  MoveL 5081 to (509.6, 509.6, 11.2) mm, rotated rx 0 ry 90 rz 0 deg; joints [-12.688, -27.246, 109.927, -16.748, -82.126, 51.332]
  Call Extruder(0.559)
  MoveL 5082 to (490.4, 509.6, 11.2) mm, rotated rx 0 ry 90 rz 0 deg; joints [-13.088, -27.603, 112.214, -17.082, -83.985, 50.809]
  MoveL 5083 to (490.4, 490.4, 11.2) mm, rotated rx 0 ry 90 rz 0 deg; joints [-11.303, -27.672, 112.704, -15.276, -84.344, 50.536]
  Call Extruder(0.199)
  MoveL 5084 to (497.23, 490.4, 11.2) mm, rotated rx 0 ry 90 rz 0 deg; joints [-11.177, -27.556, 111.894, -15.169, -83.672, 50.707]
  Call Extruder(0.010)
  MoveL 5085 to (497.58, 490.4, 11.2) mm, rotated rx 0 ry 90 rz 0 deg; joints [-11.17, -27.55, 111.853, -15.163, -83.637, 50.716]
  Call Extruder(0.007)
  MoveL 5086 to (497.58, 490.75, 11.2) mm, rotated rx 0 ry 90 rz 0 deg; joints [-11.203, -27.549, 111.844, -15.196, -83.631, 50.721]
  Call Extruder(0.035)
  MoveL 5087 to (497.57, 491.95, 11.2) mm, rotated rx 0 ry 90 rz 0 deg; joints [-11.314, -27.545, 111.816, -15.308, -83.611, 50.738]
  Call Extruder(0.007)
  MoveL 5088 to (497.58, 492.3, 11.2) mm, rotated rx 0 ry 90 rz 0 deg; joints [-11.346, -27.544, 111.808, -15.341, -83.605, 50.743]
  Set speed (120.0 mm/s)
  MoveL 5089 to (497.93, 492.3, 11.2) mm, rotated rx 0 ry 90 rz 0 deg; joints [-11.34, -27.537, 111.766, -15.336, -83.571, 50.752]
  Set speed (1000.0 mm/s)
  MoveL 5090 to (497.98, 492.3, 11.2) mm, rotated rx 0 ry 90 rz 0 deg; joints [-11.339, -27.536, 111.76, -15.335, -83.566, 50.753]
  Set speed (1000.0 mm/s)
  MoveL 5091 to (497.97, 493, 11.2) mm, rotated rx 0 ry 90 rz 0 deg; joints [-11.403, -27.534, 111.743, -15.4, -83.554, 50.764]
  Set speed (1000.0 mm/s)
  MoveL 5092 to (490.68, 490.68, 11.2) mm, rotated rx 0 ry 90 rz 0 deg; joints [-11.324, -27.666, 112.664, -15.298, -84.312, 50.546]
  Set speed (1000.0 mm/s)
  MoveL 5093 to (490.68, 490.68, 11.3) mm, rotated rx 0 ry 90 rz 0 deg; joints [-11.324, -27.677, 112.669, -15.298, -84.307, 50.548]
  Set speed (30.0 mm/s)
  Call Extruder(0.767)
  MoveL 5094 to (509.32, 509.32, 11.3) mm, rotated rx 0 ry 90 rz 0 deg; joints [-12.669, -27.264, 109.974, -16.727, -82.153, 51.321]
  MoveL 5095 to (509.44, 509.44, 11.3) mm, rotated rx 0 ry 90 rz 0 deg; joints [-12.677, -27.261, 109.956, -16.736, -82.139, 51.327]
  Set speed (120.0 mm/s)
  MoveL 5096 to (507.63, 502.27, 11.3) mm, rotated rx 0 ry 90 rz 0 deg; joints [-12.067, -27.328, 110.363, -16.108, -82.444, 51.156]
  Set speed (30.0 mm/s)
  Call Extruder(0.290)
  MoveL 5097 to (500.58, 509.32, 11.3) mm, rotated rx 0 ry 90 rz 0 deg; joints [-12.847, -27.433, 111.021, -16.874, -82.999, 51.086]
  Set speed (120.0 mm/s)
  MoveL 5098 to (499.42, 509.32, 11.3) mm, rotated rx 0 ry 90 rz 0 deg; joints [-12.872, -27.455, 111.159, -16.894, -83.111, 51.055]
  Set speed (30.0 mm/s)
  Call Extruder(0.360)
  MoveL 5099 to (490.68, 500.58, 11.3) mm, rotated rx 0 ry 90 rz 0 deg; joints [-12.247, -27.643, 112.425, -16.231, -84.127, 50.685]
  Set speed (120.0 mm/s)
  MoveL 5100 to (490.68, 499.42, 11.3) mm, rotated rx 0 ry 90 rz 0 deg; joints [-12.139, -27.647, 112.455, -16.122, -84.149, 50.668]
  Set speed (30.0 mm/s)
  Call Extruder(0.282)
  MoveL 5101 to (497.52, 492.58, 11.3) mm, rotated rx 0 ry 90 rz 0 deg; joints [-11.373, -27.554, 111.813, -15.368, -83.6, 50.747]
  MoveL 5102 to (497.64, 492.46, 11.3) mm, rotated rx 0 ry 90 rz 0 deg; joints [-11.359, -27.552, 111.801, -15.355, -83.59, 50.749]
  Set speed (120.0 mm/s)
  MoveL 5103 to (501.52, 492.33, 11.3) mm, rotated rx 0 ry 90 rz 0 deg; joints [-11.276, -27.483, 111.342, -15.283, -83.212, 50.844]
  Set speed (1000.0 mm/s)
  MoveL 5104 to (501.77, 491.87, 11.3) mm, rotated rx 0 ry 90 rz 0 deg; joints [-11.23, -27.48, 111.322, -15.237, -83.195, 50.844]
  Set speed (30.0 mm/s)
  Call Extruder(0.231)
  MoveL 5105 to (507.39, 497.49, 11.3) mm, rotated rx 0 ry 90 rz 0 deg; joints [-11.638, -27.353, 110.513, -15.671, -82.55, 51.072]
  MoveL 5106 to (507.51, 497.61, 11.3) mm, rotated rx 0 ry 90 rz 0 deg; joints [-11.647, -27.35, 110.495, -15.681, -82.536, 51.077]
  Set speed (120.0 mm/s)
  MoveL 5107 to (509.32, 490.68, 11.3) mm, rotated rx 0 ry 90 rz 0 deg; joints [-10.985, -27.341, 110.444, -15.015, -82.474, 51.011]
  Set speed (30.0 mm/s)
  Call Extruder(0.767)
  MoveL 5108 to (490.68, 509.32, 11.3) mm, rotated rx 0 ry 90 rz 0 deg; joints [-13.056, -27.61, 112.194, -17.051, -83.959, 50.814]
  MoveL 5109 to (490.56, 509.44, 11.3) mm, rotated rx 0 ry 90 rz 0 deg; joints [-13.07, -27.611, 112.205, -17.064, -83.968, 50.812]
  Set speed (120.0 mm/s)
  MoveL 5110 to (497.45, 492.37, 11.3) mm, rotated rx 0 ry 90 rz 0 deg; joints [-11.355, -27.556, 111.826, -15.35, -83.611, 50.743]
  Set speed (1000.0 mm/s)
  MoveL 5111 to (497.52, 492.3, 11.3) mm, rotated rx 0 ry 90 rz 0 deg; joints [-11.347, -27.555, 111.82, -15.342, -83.605, 50.743]
  Set speed (15.0 mm/s)
  Call Extruder(0.010)
  MoveL 5112 to (497.87, 492.3, 11.3) mm, rotated rx 0 ry 90 rz 0 deg; joints [-11.341, -27.549, 111.778, -15.337, -83.571, 50.752]
  Call Extruder(0.105)
  MoveL 5113 to (501.49, 492.3, 11.3) mm, rotated rx 0 ry 90 rz 0 deg; joints [-11.274, -27.484, 111.346, -15.281, -83.215, 50.843]
  Call Extruder(0.055)
  MoveL 5114 to (501.49, 490.4, 11.3) mm, rotated rx 0 ry 90 rz 0 deg; joints [-11.099, -27.491, 111.39, -15.104, -83.247, 50.815]
  Call Extruder(0.236)
  MoveL 5115 to (509.6, 490.4, 11.3) mm, rotated rx 0 ry 90 rz 0 deg; joints [-10.955, -27.337, 110.417, -14.985, -82.451, 51.013]
  Call Extruder(0.196)
  MoveL 5116 to (509.6, 497.15, 11.3) mm, rotated rx 0 ry 90 rz 0 deg; joints [-11.567, -27.31, 110.255, -15.607, -82.339, 51.122]
  Call Extruder(0.056)
  MoveL 5117 to (507.67, 497.15, 11.3) mm, rotated rx 0 ry 90 rz 0 deg; joints [-11.603, -27.348, 110.487, -15.636, -82.528, 51.073]
  Call Extruder(0.069)
  MoveL 5118 to (507.67, 499.52, 11.3) mm, rotated rx 0 ry 90 rz 0 deg; joints [-11.818, -27.339, 110.428, -15.854, -82.488, 51.112]
  Call Extruder(0.072)
  MoveL 5119 to (507.66, 501.99, 11.3) mm, rotated rx 0 ry 90 rz 0 deg; joints [-12.041, -27.329, 110.366, -16.082, -82.445, 51.153]
  Call Extruder(0.056)
  MoveL 5120 to (509.6, 502, 11.3) mm, rotated rx 0 ry 90 rz 0 deg; joints [-12.004, -27.29, 110.133, -16.052, -82.256, 51.203]
  Call Extruder(0.221)
  MoveL 5121 to (509.6, 509.6, 11.3) mm, rotated rx 0 ry 90 rz 0 deg; joints [-12.688, -27.257, 109.932, -16.748, -82.121, 51.334]
  Call Extruder(0.559)
  MoveL 5122 to (490.4, 509.6, 11.3) mm, rotated rx 0 ry 90 rz 0 deg; joints [-13.088, -27.613, 112.219, -17.082, -83.98, 50.811]
  MoveL 5123 to (490.4, 490.4, 11.3) mm, rotated rx 0 ry 90 rz 0 deg; joints [-11.303, -27.682, 112.709, -15.277, -84.339, 50.537]
  Call Extruder(0.197)
  MoveL 5124 to (497.17, 490.4, 11.3) mm, rotated rx 0 ry 90 rz 0 deg; joints [-11.178, -27.568, 111.906, -15.17, -83.672, 50.708]
  Call Extruder(0.010)
  MoveL 5125 to (497.52, 490.4, 11.3) mm, rotated rx 0 ry 90 rz 0 deg; joints [-11.171, -27.562, 111.864, -15.164, -83.638, 50.716]
  Call Extruder(0.007)
  MoveL 5126 to (497.52, 490.75, 11.3) mm, rotated rx 0 ry 90 rz 0 deg; joints [-11.204, -27.561, 111.856, -15.197, -83.632, 50.721]
  Call Extruder(0.035)
  MoveL 5127 to (497.52, 491.95, 11.3) mm, rotated rx 0 ry 90 rz 0 deg; joints [-11.315, -27.556, 111.828, -15.309, -83.611, 50.738]
  Call Extruder(0.007)
  MoveL 5128 to (497.52, 492.3, 11.3) mm, rotated rx 0 ry 90 rz 0 deg; joints [-11.347, -27.555, 111.82, -15.342, -83.605, 50.743]
  Set speed (120.0 mm/s)
  MoveL 5129 to (497.87, 492.3, 11.3) mm, rotated rx 0 ry 90 rz 0 deg; joints [-11.341, -27.549, 111.778, -15.337, -83.571, 50.752]
  Set speed (1000.0 mm/s)
  MoveL 5130 to (497.92, 492.3, 11.3) mm, rotated rx 0 ry 90 rz 0 deg; joints [-11.34, -27.548, 111.772, -15.336, -83.566, 50.753]
  Set speed (1000.0 mm/s)
  MoveL 5131 to (497.92, 493, 11.3) mm, rotated rx 0 ry 90 rz 0 deg; joints [-11.404, -27.546, 111.755, -15.401, -83.554, 50.764]
  Set speed (1000.0 mm/s)
  MoveL 5132 to (490.68, 490.68, 11.3) mm, rotated rx 0 ry 90 rz 0 deg; joints [-11.324, -27.677, 112.669, -15.298, -84.307, 50.548]
  Set speed (1000.0 mm/s)
  MoveL 5133 to (490.68, 490.68, 11.4) mm, rotated rx 0 ry 90 rz 0 deg; joints [-11.324, -27.688, 112.675, -15.299, -84.301, 50.549]
  Set speed (30.0 mm/s)
  Call Extruder(0.767)
  MoveL 5134 to (509.32, 509.32, 11.4) mm, rotated rx 0 ry 90 rz 0 deg; joints [-12.669, -27.274, 109.979, -16.727, -82.148, 51.323]
  MoveL 5135 to (509.44, 509.44, 11.4) mm, rotated rx 0 ry 90 rz 0 deg; joints [-12.677, -27.271, 109.961, -16.736, -82.134, 51.328]
  Set speed (120.0 mm/s)
  MoveL 5136 to (507.57, 502.33, 11.4) mm, rotated rx 0 ry 90 rz 0 deg; joints [-12.073, -27.34, 110.374, -16.114, -82.443, 51.157]
  Set speed (30.0 mm/s)
  Call Extruder(0.288)
  MoveL 5137 to (500.58, 509.32, 11.4) mm, rotated rx 0 ry 90 rz 0 deg; joints [-12.847, -27.444, 111.026, -16.874, -82.994, 51.088]
  Set speed (120.0 mm/s)
  MoveL 5138 to (499.42, 509.32, 11.4) mm, rotated rx 0 ry 90 rz 0 deg; joints [-12.872, -27.465, 111.164, -16.894, -83.106, 51.056]
  Set speed (30.0 mm/s)
  Call Extruder(0.360)
  MoveL 5139 to (490.68, 500.58, 11.4) mm, rotated rx 0 ry 90 rz 0 deg; joints [-12.247, -27.653, 112.431, -16.231, -84.122, 50.686]
  Set speed (120.0 mm/s)
  MoveL 5140 to (490.68, 499.42, 11.4) mm, rotated rx 0 ry 90 rz 0 deg; joints [-12.139, -27.658, 112.46, -16.122, -84.144, 50.67]
  Set speed (30.0 mm/s)
  Call Extruder(0.282)
  MoveL 5141 to (497.52, 492.58, 11.4) mm, rotated rx 0 ry 90 rz 0 deg; joints [-11.373, -27.565, 111.818, -15.368, -83.595, 50.749]
  MoveL 5142 to (497.64, 492.46, 11.4) mm, rotated rx 0 ry 90 rz 0 deg; joints [-11.359, -27.563, 111.806, -15.355, -83.585, 50.75]
  Set speed (120.0 mm/s)
  MoveL 5143 to (501.59, 492.33, 11.4) mm, rotated rx 0 ry 90 rz 0 deg; joints [-11.275, -27.493, 111.339, -15.282, -83.2, 50.847]
  Set speed (1000.0 mm/s)
  MoveL 5144 to (501.84, 491.94, 11.4) mm, rotated rx 0 ry 90 rz 0 deg; joints [-11.234, -27.489, 111.318, -15.242, -83.182, 50.848]
  Set speed (30.0 mm/s)
  Call Extruder(0.228)
  MoveL 5145 to (507.39, 497.49, 11.4) mm, rotated rx 0 ry 90 rz 0 deg; joints [-11.638, -27.363, 110.518, -15.671, -82.545, 51.073]
  MoveL 5146 to (507.51, 497.61, 11.4) mm, rotated rx 0 ry 90 rz 0 deg; joints [-11.647, -27.36, 110.5, -15.681, -82.531, 51.078]
  Set speed (120.0 mm/s)
  MoveL 5147 to (509.32, 490.68, 11.4) mm, rotated rx 0 ry 90 rz 0 deg; joints [-10.985, -27.352, 110.449, -15.015, -82.469, 51.012]
  Set speed (30.0 mm/s)
  Call Extruder(0.767)
  MoveL 5148 to (490.68, 509.32, 11.4) mm, rotated rx 0 ry 90 rz 0 deg; joints [-13.056, -27.62, 112.199, -17.051, -83.953, 50.816]
  MoveL 5149 to (490.56, 509.44, 11.4) mm, rotated rx 0 ry 90 rz 0 deg; joints [-13.07, -27.622, 112.21, -17.065, -83.963, 50.814]
  Set speed (120.0 mm/s)
  MoveL 5150 to (507.6, 499.64, 11.4) mm, rotated rx 0 ry 90 rz 0 deg; joints [-11.83, -27.35, 110.439, -15.867, -82.487, 51.114]
  Set speed (1000.0 mm/s)
  MoveL 5151 to (507.67, 499.57, 11.4) mm, rotated rx 0 ry 90 rz 0 deg; joints [-11.822, -27.349, 110.432, -15.859, -82.482, 51.114]
  Set speed (15.0 mm/s)
  Call Extruder(0.010)
  MoveL 5152 to (508.02, 499.57, 11.4) mm, rotated rx 0 ry 90 rz 0 deg; joints [-11.816, -27.342, 110.39, -15.854, -82.447, 51.123]
  Call Extruder(0.046)
  MoveL 5153 to (509.6, 499.57, 11.4) mm, rotated rx 0 ry 90 rz 0 deg; joints [-11.786, -27.311, 110.2, -15.829, -82.293, 51.163]
  Call Extruder(0.000)
  MoveL 5154 to (509.6, 499.58, 11.4) mm, rotated rx 0 ry 90 rz 0 deg; joints [-11.786, -27.311, 110.199, -15.83, -82.293, 51.164]
  Call Extruder(0.046)
  MoveL 5155 to (508.02, 499.58, 11.4) mm, rotated rx 0 ry 90 rz 0 deg; joints [-11.816, -27.342, 110.39, -15.854, -82.447, 51.123]
  Call Extruder(0.010)
  MoveL 5156 to (507.67, 499.58, 11.4) mm, rotated rx 0 ry 90 rz 0 deg; joints [-11.823, -27.349, 110.432, -15.86, -82.482, 51.114]
  Call Extruder(0.007)
  MoveL 5157 to (507.67, 499.93, 11.4) mm, rotated rx 0 ry 90 rz 0 deg; joints [-11.854, -27.348, 110.423, -15.892, -82.475, 51.12]
  Call Extruder(0.062)
  MoveL 5158 to (507.66, 502.05, 11.4) mm, rotated rx 0 ry 90 rz 0 deg; joints [-12.046, -27.339, 110.37, -16.087, -82.439, 51.155]
  Call Extruder(0.056)
  MoveL 5159 to (509.6, 502.05, 11.4) mm, rotated rx 0 ry 90 rz 0 deg; joints [-12.009, -27.301, 110.137, -16.057, -82.25, 51.205]
  Call Extruder(0.220)
  MoveL 5160 to (509.6, 509.6, 11.4) mm, rotated rx 0 ry 90 rz 0 deg; joints [-12.688, -27.267, 109.938, -16.748, -82.115, 51.335]
  Call Extruder(0.559)
  MoveL 5161 to (490.4, 509.6, 11.4) mm, rotated rx 0 ry 90 rz 0 deg; joints [-13.088, -27.624, 112.224, -17.082, -83.975, 50.812]
  MoveL 5162 to (490.4, 490.4, 11.4) mm, rotated rx 0 ry 90 rz 0 deg; joints [-11.303, -27.693, 112.714, -15.277, -84.334, 50.538]
  Call Extruder(0.195)
  MoveL 5163 to (497.11, 490.4, 11.4) mm, rotated rx 0 ry 90 rz 0 deg; joints [-11.179, -27.58, 111.918, -15.171, -83.672, 50.708]
  Call Extruder(0.010)
  MoveL 5164 to (497.46, 490.4, 11.4) mm, rotated rx 0 ry 90 rz 0 deg; joints [-11.172, -27.573, 111.876, -15.165, -83.638, 50.716]
  Call Extruder(0.007)
  MoveL 5165 to (497.46, 490.75, 11.4) mm, rotated rx 0 ry 90 rz 0 deg; joints [-11.205, -27.572, 111.868, -15.198, -83.632, 50.721]
  Call Extruder(0.035)
  MoveL 5166 to (497.46, 491.95, 11.4) mm, rotated rx 0 ry 90 rz 0 deg; joints [-11.316, -27.568, 111.84, -15.31, -83.612, 50.738]
  Call Extruder(0.010)
  MoveL 5167 to (497.46, 492.3, 11.4) mm, rotated rx 0 ry 90 rz 0 deg; joints [-11.348, -27.567, 111.831, -15.343, -83.606, 50.743]
  Call Extruder(0.007)
  MoveL 5168 to (497.81, 492.3, 11.4) mm, rotated rx 0 ry 90 rz 0 deg; joints [-11.342, -27.561, 111.79, -15.338, -83.571, 50.752]
  Call Extruder(0.109)
  MoveL 5169 to (501.56, 492.3, 11.4) mm, rotated rx 0 ry 90 rz 0 deg; joints [-11.272, -27.493, 111.343, -15.28, -83.203, 50.846]
  Call Extruder(0.055)
  MoveL 5170 to (501.56, 490.4, 11.4) mm, rotated rx 0 ry 90 rz 0 deg; joints [-11.098, -27.5, 111.388, -15.103, -83.235, 50.818]
  Call Extruder(0.234)
  MoveL 5171 to (509.6, 490.4, 11.4) mm, rotated rx 0 ry 90 rz 0 deg; joints [-10.955, -27.347, 110.422, -14.985, -82.445, 51.015]
  Call Extruder(0.195)
  MoveL 5172 to (509.6, 497.09, 11.4) mm, rotated rx 0 ry 90 rz 0 deg; joints [-11.561, -27.321, 110.261, -15.601, -82.335, 51.122]
  Call Extruder(0.056)
  MoveL 5173 to (507.67, 497.09, 11.4) mm, rotated rx 0 ry 90 rz 0 deg; joints [-11.597, -27.359, 110.494, -15.631, -82.524, 51.074]
  Call Extruder(0.062)
  MoveL 5174 to (507.67, 499.22, 11.4) mm, rotated rx 0 ry 90 rz 0 deg; joints [-11.79, -27.351, 110.441, -15.827, -82.488, 51.108]
  Call Extruder(0.007)
  MoveL 5175 to (507.67, 499.57, 11.4) mm, rotated rx 0 ry 90 rz 0 deg; joints [-11.822, -27.349, 110.432, -15.859, -82.482, 51.114]
  Set speed (120.0 mm/s)
  MoveL 5176 to (508.02, 499.57, 11.4) mm, rotated rx 0 ry 90 rz 0 deg; joints [-11.816, -27.342, 110.39, -15.854, -82.447, 51.123]
  Set speed (1000.0 mm/s)
  MoveL 5177 to (508.07, 499.57, 11.4) mm, rotated rx 0 ry 90 rz 0 deg; joints [-11.815, -27.341, 110.384, -15.853, -82.443, 51.124]
  Set speed (1000.0 mm/s)
  MoveL 5178 to (506.97, 500.27, 11.4) mm, rotated rx 0 ry 90 rz 0 deg; joints [-11.899, -27.36, 110.499, -15.934, -82.538, 51.108]
  Set speed (1000.0 mm/s)
  MoveL 5179 to (490.68, 490.68, 11.4) mm, rotated rx 0 ry 90 rz 0 deg; joints [-11.324, -27.688, 112.675, -15.299, -84.301, 50.549]
  Set speed (1000.0 mm/s)
  MoveL 5180 to (490.68, 490.68, 11.5) mm, rotated rx 0 ry 90 rz 0 deg; joints [-11.324, -27.698, 112.68, -15.299, -84.296, 50.551]
  Set speed (30.0 mm/s)
  Call Extruder(0.767)
  MoveL 5181 to (509.32, 509.32, 11.5) mm, rotated rx 0 ry 90 rz 0 deg; joints [-12.669, -27.285, 109.984, -16.727, -82.143, 51.324]
  MoveL 5182 to (509.44, 509.44, 11.5) mm, rotated rx 0 ry 90 rz 0 deg; joints [-12.677, -27.282, 109.966, -16.737, -82.129, 51.33]
  Set speed (120.0 mm/s)
  MoveL 5183 to (507.51, 502.39, 11.5) mm, rotated rx 0 ry 90 rz 0 deg; joints [-12.08, -27.351, 110.384, -16.121, -82.442, 51.158]
  Set speed (30.0 mm/s)
  Call Extruder(0.285)
  MoveL 5184 to (500.58, 509.32, 11.5) mm, rotated rx 0 ry 90 rz 0 deg; joints [-12.847, -27.454, 111.031, -16.874, -82.988, 51.089]
  Set speed (120.0 mm/s)
  MoveL 5185 to (499.42, 509.32, 11.5) mm, rotated rx 0 ry 90 rz 0 deg; joints [-12.872, -27.476, 111.169, -16.895, -83.101, 51.058]
  Set speed (30.0 mm/s)
  Call Extruder(0.360)
  MoveL 5186 to (490.68, 500.58, 11.5) mm, rotated rx 0 ry 90 rz 0 deg; joints [-12.247, -27.664, 112.436, -16.232, -84.117, 50.688]
  Set speed (120.0 mm/s)
  MoveL 5187 to (490.68, 499.42, 11.5) mm, rotated rx 0 ry 90 rz 0 deg; joints [-12.139, -27.668, 112.465, -16.123, -84.138, 50.671]
  Set speed (30.0 mm/s)
  Call Extruder(0.282)
  MoveL 5188 to (497.52, 492.58, 11.5) mm, rotated rx 0 ry 90 rz 0 deg; joints [-11.373, -27.575, 111.823, -15.368, -83.59, 50.75]
  MoveL 5189 to (497.64, 492.46, 11.5) mm, rotated rx 0 ry 90 rz 0 deg; joints [-11.359, -27.574, 111.811, -15.355, -83.58, 50.752]
  Set speed (120.0 mm/s)
  MoveL 5190 to (501.65, 492.33, 11.5) mm, rotated rx 0 ry 90 rz 0 deg; joints [-11.273, -27.502, 111.337, -15.281, -83.189, 50.85]
  Set speed (1000.0 mm/s)
  MoveL 5191 to (501.9, 492, 11.5) mm, rotated rx 0 ry 90 rz 0 deg; joints [-11.239, -27.498, 111.314, -15.247, -83.17, 50.852]
  Set speed (30.0 mm/s)
  Call Extruder(0.226)
  MoveL 5192 to (507.39, 497.49, 11.5) mm, rotated rx 0 ry 90 rz 0 deg; joints [-11.638, -27.374, 110.523, -15.672, -82.54, 51.075]
  MoveL 5193 to (507.51, 497.61, 11.5) mm, rotated rx 0 ry 90 rz 0 deg; joints [-11.647, -27.371, 110.506, -15.681, -82.526, 51.08]
  Set speed (120.0 mm/s)
  MoveL 5194 to (509.32, 490.68, 11.5) mm, rotated rx 0 ry 90 rz 0 deg; joints [-10.985, -27.362, 110.454, -15.015, -82.463, 51.014]
  Set speed (30.0 mm/s)
  Call Extruder(0.767)
  MoveL 5195 to (490.68, 509.32, 11.5) mm, rotated rx 0 ry 90 rz 0 deg; joints [-13.056, -27.631, 112.204, -17.051, -83.948, 50.817]
  MoveL 5196 to (490.56, 509.44, 11.5) mm, rotated rx 0 ry 90 rz 0 deg; joints [-13.07, -27.633, 112.216, -17.065, -83.958, 50.816]
  Set speed (120.0 mm/s)
  MoveL 5197 to (507.6, 499.56, 11.5) mm, rotated rx 0 ry 90 rz 0 deg; joints [-11.823, -27.361, 110.446, -15.86, -82.484, 51.114]
  Set speed (1000.0 mm/s)
  MoveL 5198 to (507.67, 499.63, 11.5) mm, rotated rx 0 ry 90 rz 0 deg; joints [-11.828, -27.359, 110.436, -15.865, -82.476, 51.117]
  Set speed (15.0 mm/s)
  Call Extruder(0.010)
  MoveL 5199 to (507.67, 499.98, 11.5) mm, rotated rx 0 ry 90 rz 0 deg; joints [-11.859, -27.358, 110.427, -15.897, -82.469, 51.122]
  Call Extruder(0.062)
  MoveL 5200 to (507.67, 502.11, 11.5) mm, rotated rx 0 ry 90 rz 0 deg; joints [-12.051, -27.349, 110.373, -16.092, -82.432, 51.157]
  Call Extruder(0.056)
  MoveL 5201 to (509.6, 502.11, 11.5) mm, rotated rx 0 ry 90 rz 0 deg; joints [-12.015, -27.311, 110.14, -16.063, -82.244, 51.207]
  Call Extruder(0.218)
  MoveL 5202 to (509.6, 509.6, 11.5) mm, rotated rx 0 ry 90 rz 0 deg; joints [-12.688, -27.278, 109.943, -16.748, -82.11, 51.337]
  Call Extruder(0.559)
  MoveL 5203 to (490.4, 509.6, 11.5) mm, rotated rx 0 ry 90 rz 0 deg; joints [-13.088, -27.635, 112.23, -17.082, -83.97, 50.814]
  MoveL 5204 to (490.4, 490.4, 11.5) mm, rotated rx 0 ry 90 rz 0 deg; joints [-11.303, -27.704, 112.719, -15.277, -84.329, 50.54]
  Call Extruder(0.204)
  MoveL 5205 to (497.41, 490.4, 11.5) mm, rotated rx 0 ry 90 rz 0 deg; joints [-11.173, -27.585, 111.888, -15.166, -83.638, 50.716]
  Call Extruder(0.045)
  MoveL 5206 to (497.41, 491.95, 11.5) mm, rotated rx 0 ry 90 rz 0 deg; joints [-11.317, -27.58, 111.852, -15.311, -83.612, 50.738]
  Call Extruder(0.010)
  MoveL 5207 to (497.41, 492.3, 11.5) mm, rotated rx 0 ry 90 rz 0 deg; joints [-11.349, -27.578, 111.843, -15.344, -83.606, 50.743]
  Call Extruder(0.007)
  MoveL 5208 to (497.76, 492.3, 11.5) mm, rotated rx 0 ry 90 rz 0 deg; joints [-11.343, -27.572, 111.802, -15.339, -83.571, 50.752]
  Call Extruder(0.112)
  MoveL 5209 to (501.62, 492.3, 11.5) mm, rotated rx 0 ry 90 rz 0 deg; joints [-11.271, -27.503, 111.341, -15.279, -83.192, 50.849]
  Call Extruder(0.055)
  MoveL 5210 to (501.62, 490.4, 11.5) mm, rotated rx 0 ry 90 rz 0 deg; joints [-11.097, -27.509, 111.385, -15.102, -83.224, 50.821]
  Call Extruder(0.232)
  MoveL 5211 to (509.6, 490.4, 11.5) mm, rotated rx 0 ry 90 rz 0 deg; joints [-10.955, -27.358, 110.427, -14.985, -82.44, 51.016]
  Call Extruder(0.193)
  MoveL 5212 to (509.6, 497.03, 11.5) mm, rotated rx 0 ry 90 rz 0 deg; joints [-11.556, -27.332, 110.268, -15.596, -82.331, 51.123]
  Call Extruder(0.056)
  MoveL 5213 to (507.67, 497.03, 11.5) mm, rotated rx 0 ry 90 rz 0 deg; joints [-11.592, -27.37, 110.501, -15.626, -82.52, 51.074]
  Call Extruder(0.062)
  MoveL 5214 to (507.67, 499.16, 11.5) mm, rotated rx 0 ry 90 rz 0 deg; joints [-11.785, -27.361, 110.448, -15.822, -82.483, 51.109]
  Call Extruder(0.010)
  MoveL 5215 to (507.67, 499.51, 11.5) mm, rotated rx 0 ry 90 rz 0 deg; joints [-11.817, -27.36, 110.439, -15.854, -82.477, 51.115]
  Call Extruder(0.007)
  MoveL 5216 to (508.02, 499.51, 11.5) mm, rotated rx 0 ry 90 rz 0 deg; joints [-11.81, -27.353, 110.397, -15.849, -82.443, 51.124]
  Call Extruder(0.046)
  MoveL 5217 to (509.6, 499.51, 11.5) mm, rotated rx 0 ry 90 rz 0 deg; joints [-11.78, -27.322, 110.206, -15.824, -82.289, 51.164]
  Call Extruder(0.004)
  MoveL 5218 to (509.6, 499.64, 11.5) mm, rotated rx 0 ry 90 rz 0 deg; joints [-11.792, -27.321, 110.203, -15.836, -82.287, 51.166]
  Call Extruder(0.046)
  MoveL 5219 to (508.02, 499.63, 11.5) mm, rotated rx 0 ry 90 rz 0 deg; joints [-11.821, -27.352, 110.394, -15.86, -82.441, 51.126]
  Call Extruder(0.007)
  MoveL 5220 to (507.67, 499.63, 11.5) mm, rotated rx 0 ry 90 rz 0 deg; joints [-11.828, -27.359, 110.436, -15.865, -82.476, 51.117]
  Set speed (120.0 mm/s)
  MoveL 5221 to (507.67, 499.98, 11.5) mm, rotated rx 0 ry 90 rz 0 deg; joints [-11.859, -27.358, 110.427, -15.897, -82.469, 51.122]
  Set speed (1000.0 mm/s)
  MoveL 5222 to (507.67, 500.03, 11.5) mm, rotated rx 0 ry 90 rz 0 deg; joints [-11.864, -27.358, 110.426, -15.902, -82.469, 51.123]
  Set speed (1000.0 mm/s)
  MoveL 5223 to (506.97, 500.03, 11.5) mm, rotated rx 0 ry 90 rz 0 deg; joints [-11.877, -27.371, 110.51, -15.913, -82.537, 51.105]
  Set speed (1000.0 mm/s)
  MoveL 5224 to (490.68, 490.68, 11.5) mm, rotated rx 0 ry 90 rz 0 deg; joints [-11.324, -27.698, 112.68, -15.299, -84.296, 50.551]
  Set speed (1000.0 mm/s)
  MoveL 5225 to (490.68, 490.68, 11.6) mm, rotated rx 0 ry 90 rz 0 deg; joints [-11.324, -27.709, 112.685, -15.299, -84.291, 50.552]
  Set speed (30.0 mm/s)
  Call Extruder(0.767)
  MoveL 5226 to (509.32, 509.32, 11.6) mm, rotated rx 0 ry 90 rz 0 deg; joints [-12.669, -27.295, 109.989, -16.728, -82.138, 51.326]
  MoveL 5227 to (509.44, 509.44, 11.6) mm, rotated rx 0 ry 90 rz 0 deg; joints [-12.677, -27.292, 109.971, -16.737, -82.123, 51.331]
  Set speed (120.0 mm/s)
  MoveL 5228 to (507.46, 502.44, 11.6) mm, rotated rx 0 ry 90 rz 0 deg; joints [-12.086, -27.362, 110.395, -16.127, -82.442, 51.159]
  Set speed (30.0 mm/s)
  Call Extruder(0.283)
  MoveL 5229 to (500.58, 509.32, 11.6) mm, rotated rx 0 ry 90 rz 0 deg; joints [-12.847, -27.465, 111.036, -16.875, -82.983, 51.091]
  Set speed (120.0 mm/s)
  MoveL 5230 to (499.42, 509.32, 11.6) mm, rotated rx 0 ry 90 rz 0 deg; joints [-12.872, -27.487, 111.174, -16.895, -83.096, 51.059]
  Set speed (30.0 mm/s)
  Call Extruder(0.360)
  MoveL 5231 to (490.68, 500.58, 11.6) mm, rotated rx 0 ry 90 rz 0 deg; joints [-12.247, -27.675, 112.441, -16.232, -84.112, 50.689]
  Set speed (120.0 mm/s)
  MoveL 5232 to (490.68, 499.42, 11.6) mm, rotated rx 0 ry 90 rz 0 deg; joints [-12.139, -27.679, 112.471, -16.123, -84.133, 50.673]
  Set speed (30.0 mm/s)
  Call Extruder(0.282)
  MoveL 5233 to (497.52, 492.58, 11.6) mm, rotated rx 0 ry 90 rz 0 deg; joints [-11.373, -27.586, 111.828, -15.369, -83.585, 50.752]
  MoveL 5234 to (497.64, 492.46, 11.6) mm, rotated rx 0 ry 90 rz 0 deg; joints [-11.359, -27.584, 111.817, -15.355, -83.575, 50.753]
  Set speed (120.0 mm/s)
  MoveL 5235 to (501.71, 492.33, 11.6) mm, rotated rx 0 ry 90 rz 0 deg; joints [-11.272, -27.511, 111.334, -15.28, -83.177, 50.853]
  Set speed (1000.0 mm/s)
  MoveL 5236 to (501.96, 492.06, 11.6) mm, rotated rx 0 ry 90 rz 0 deg; joints [-11.244, -27.508, 111.31, -15.252, -83.157, 50.856]
  Set speed (30.0 mm/s)
  Call Extruder(0.223)
  MoveL 5237 to (507.39, 497.49, 11.6) mm, rotated rx 0 ry 90 rz 0 deg; joints [-11.638, -27.384, 110.528, -15.672, -82.534, 51.076]
  MoveL 5238 to (507.51, 497.61, 11.6) mm, rotated rx 0 ry 90 rz 0 deg; joints [-11.647, -27.381, 110.51, -15.681, -82.52, 51.081]
  Set speed (120.0 mm/s)
  MoveL 5239 to (509.32, 490.68, 11.6) mm, rotated rx 0 ry 90 rz 0 deg; joints [-10.985, -27.373, 110.46, -15.015, -82.458, 51.015]
  Set speed (30.0 mm/s)
  Call Extruder(0.767)
  MoveL 5240 to (490.68, 509.32, 11.6) mm, rotated rx 0 ry 90 rz 0 deg; joints [-13.056, -27.642, 112.21, -17.051, -83.943, 50.819]
  MoveL 5241 to (490.56, 509.44, 11.6) mm, rotated rx 0 ry 90 rz 0 deg; joints [-13.07, -27.643, 112.221, -17.065, -83.952, 50.817]
  Set speed (120.0 mm/s)
  MoveL 5242 to (507.6, 499.52, 11.6) mm, rotated rx 0 ry 90 rz 0 deg; joints [-11.819, -27.372, 110.452, -15.856, -82.479, 51.115]
  Set speed (1000.0 mm/s)
  MoveL 5243 to (507.67, 499.46, 11.6) mm, rotated rx 0 ry 90 rz 0 deg; joints [-11.812, -27.371, 110.445, -15.849, -82.473, 51.115]
  Set speed (15.0 mm/s)
  Call Extruder(0.010)
  MoveL 5244 to (508.02, 499.45, 11.6) mm, rotated rx 0 ry 90 rz 0 deg; joints [-11.805, -27.364, 110.404, -15.843, -82.439, 51.124]
  Call Extruder(0.046)
  MoveL 5245 to (509.6, 499.45, 11.6) mm, rotated rx 0 ry 90 rz 0 deg; joints [-11.775, -27.332, 110.213, -15.819, -82.285, 51.164]
  Call Extruder(0.007)
  MoveL 5246 to (509.6, 499.69, 11.6) mm, rotated rx 0 ry 90 rz 0 deg; joints [-11.796, -27.331, 110.207, -15.841, -82.281, 51.168]
  Call Extruder(0.031)
  MoveL 5247 to (508.02, 499.69, 11.6) mm, rotated rx 0 ry 90 rz 0 deg; joints [-11.826, -27.363, 110.398, -15.865, -82.435, 51.128]
  Call Extruder(0.007)
  MoveL 5248 to (507.67, 499.69, 11.6) mm, rotated rx 0 ry 90 rz 0 deg; joints [-11.833, -27.37, 110.44, -15.87, -82.469, 51.119]
  Call Extruder(0.007)
  MoveL 5249 to (507.67, 500.04, 11.6) mm, rotated rx 0 ry 90 rz 0 deg; joints [-11.865, -27.368, 110.431, -15.903, -82.463, 51.125]
  Call Extruder(0.062)
  MoveL 5250 to (507.67, 502.16, 11.6) mm, rotated rx 0 ry 90 rz 0 deg; joints [-12.057, -27.359, 110.377, -16.098, -82.426, 51.16]
  Call Extruder(0.056)
  MoveL 5251 to (509.6, 502.17, 11.6) mm, rotated rx 0 ry 90 rz 0 deg; joints [-12.02, -27.321, 110.144, -16.068, -82.238, 51.21]
  Call Extruder(0.216)
  MoveL 5252 to (509.6, 509.6, 11.6) mm, rotated rx 0 ry 90 rz 0 deg; joints [-12.688, -27.288, 109.948, -16.749, -82.105, 51.338]
  Call Extruder(0.559)
  MoveL 5253 to (490.4, 509.6, 11.6) mm, rotated rx 0 ry 90 rz 0 deg; joints [-13.088, -27.645, 112.235, -17.083, -83.964, 50.815]
  MoveL 5254 to (490.4, 490.4, 11.6) mm, rotated rx 0 ry 90 rz 0 deg; joints [-11.303, -27.715, 112.725, -15.277, -84.323, 50.541]
  Call Extruder(0.192)
  MoveL 5255 to (497, 490.4, 11.6) mm, rotated rx 0 ry 90 rz 0 deg; joints [-11.181, -27.603, 111.942, -15.173, -83.673, 50.708]
  Call Extruder(0.010)
  MoveL 5256 to (497.35, 490.4, 11.6) mm, rotated rx 0 ry 90 rz 0 deg; joints [-11.175, -27.597, 111.9, -15.167, -83.639, 50.716]
  Call Extruder(0.007)
  MoveL 5257 to (497.35, 490.75, 11.6) mm, rotated rx 0 ry 90 rz 0 deg; joints [-11.207, -27.595, 111.892, -15.2, -83.633, 50.721]
  Call Extruder(0.035)
  MoveL 5258 to (497.35, 491.95, 11.6) mm, rotated rx 0 ry 90 rz 0 deg; joints [-11.318, -27.591, 111.864, -15.312, -83.612, 50.738]
  Call Extruder(0.010)
  MoveL 5259 to (497.35, 492.3, 11.6) mm, rotated rx 0 ry 90 rz 0 deg; joints [-11.35, -27.59, 111.855, -15.345, -83.606, 50.743]
  Call Extruder(0.007)
  MoveL 5260 to (497.7, 492.3, 11.6) mm, rotated rx 0 ry 90 rz 0 deg; joints [-11.344, -27.584, 111.814, -15.34, -83.572, 50.752]
  Call Extruder(0.116)
  MoveL 5261 to (501.68, 492.3, 11.6) mm, rotated rx 0 ry 90 rz 0 deg; joints [-11.27, -27.512, 111.338, -15.278, -83.18, 50.852]
  Call Extruder(0.055)
  MoveL 5262 to (501.68, 490.4, 11.6) mm, rotated rx 0 ry 90 rz 0 deg; joints [-11.096, -27.519, 111.383, -15.101, -83.212, 50.824]
  Call Extruder(0.230)
  MoveL 5263 to (509.6, 490.4, 11.6) mm, rotated rx 0 ry 90 rz 0 deg; joints [-10.955, -27.368, 110.432, -14.986, -82.435, 51.018]
  Call Extruder(0.191)
  MoveL 5264 to (509.6, 496.97, 11.6) mm, rotated rx 0 ry 90 rz 0 deg; joints [-11.551, -27.343, 110.275, -15.591, -82.327, 51.123]
  Call Extruder(0.056)
  MoveL 5265 to (507.67, 496.97, 11.6) mm, rotated rx 0 ry 90 rz 0 deg; joints [-11.587, -27.381, 110.507, -15.62, -82.516, 51.075]
  Call Extruder(0.062)
  MoveL 5266 to (507.67, 499.11, 11.6) mm, rotated rx 0 ry 90 rz 0 deg; joints [-11.78, -27.372, 110.454, -15.817, -82.479, 51.11]
  Call Extruder(0.007)
  MoveL 5267 to (507.67, 499.46, 11.6) mm, rotated rx 0 ry 90 rz 0 deg; joints [-11.812, -27.371, 110.445, -15.849, -82.473, 51.115]
  Set speed (120.0 mm/s)
  MoveL 5268 to (508.02, 499.45, 11.6) mm, rotated rx 0 ry 90 rz 0 deg; joints [-11.805, -27.364, 110.404, -15.843, -82.439, 51.124]
  Set speed (1000.0 mm/s)
  MoveL 5269 to (508.07, 499.45, 11.6) mm, rotated rx 0 ry 90 rz 0 deg; joints [-11.804, -27.363, 110.397, -15.843, -82.434, 51.125]
  Set speed (1000.0 mm/s)
  MoveL 5270 to (506.97, 500.15, 11.6) mm, rotated rx 0 ry 90 rz 0 deg; joints [-11.888, -27.381, 110.512, -15.924, -82.53, 51.109]
  Set speed (1000.0 mm/s)
  MoveL 5271 to (490.68, 490.68, 11.6) mm, rotated rx 0 ry 90 rz 0 deg; joints [-11.324, -27.709, 112.685, -15.299, -84.291, 50.552]
  Set speed (1000.0 mm/s)
  MoveL 5272 to (490.68, 490.68, 11.7) mm, rotated rx 0 ry 90 rz 0 deg; joints [-11.324, -27.72, 112.69, -15.299, -84.286, 50.554]
  Set speed (30.0 mm/s)
  Call Extruder(0.767)
  MoveL 5273 to (509.32, 509.32, 11.7) mm, rotated rx 0 ry 90 rz 0 deg; joints [-12.669, -27.306, 109.994, -16.728, -82.133, 51.327]
  MoveL 5274 to (509.44, 509.44, 11.7) mm, rotated rx 0 ry 90 rz 0 deg; joints [-12.677, -27.303, 109.976, -16.737, -82.118, 51.333]
  Set speed (120.0 mm/s)
  MoveL 5275 to (507.4, 502.5, 11.7) mm, rotated rx 0 ry 90 rz 0 deg; joints [-12.092, -27.374, 110.405, -16.133, -82.441, 51.16]
  Set speed (30.0 mm/s)
  Call Extruder(0.281)
  MoveL 5276 to (500.58, 509.32, 11.7) mm, rotated rx 0 ry 90 rz 0 deg; joints [-12.847, -27.476, 111.041, -16.875, -82.978, 51.092]
  Set speed (120.0 mm/s)
  MoveL 5277 to (499.42, 509.32, 11.7) mm, rotated rx 0 ry 90 rz 0 deg; joints [-12.872, -27.497, 111.179, -16.895, -83.09, 51.061]
  Set speed (30.0 mm/s)
  Call Extruder(0.360)
  MoveL 5278 to (490.68, 500.58, 11.7) mm, rotated rx 0 ry 90 rz 0 deg; joints [-12.247, -27.685, 112.446, -16.232, -84.106, 50.691]
  Set speed (120.0 mm/s)
  MoveL 5279 to (490.68, 499.42, 11.7) mm, rotated rx 0 ry 90 rz 0 deg; joints [-12.139, -27.69, 112.476, -16.123, -84.128, 50.674]
  Set speed (30.0 mm/s)
  Call Extruder(0.282)
  MoveL 5280 to (497.52, 492.58, 11.7) mm, rotated rx 0 ry 90 rz 0 deg; joints [-11.373, -27.597, 111.833, -15.369, -83.579, 50.753]
  MoveL 5281 to (497.64, 492.46, 11.7) mm, rotated rx 0 ry 90 rz 0 deg; joints [-11.359, -27.595, 111.822, -15.355, -83.569, 50.755]
  Set speed (120.0 mm/s)
  MoveL 5282 to (501.78, 492.33, 11.7) mm, rotated rx 0 ry 90 rz 0 deg; joints [-11.271, -27.521, 111.332, -15.28, -83.166, 50.856]
  Set speed (1000.0 mm/s)
  MoveL 5283 to (502.03, 492.13, 11.7) mm, rotated rx 0 ry 90 rz 0 deg; joints [-11.248, -27.517, 111.306, -15.257, -83.145, 50.859]
  Set speed (30.0 mm/s)
  Call Extruder(0.221)
  MoveL 5284 to (507.39, 497.49, 11.7) mm, rotated rx 0 ry 90 rz 0 deg; joints [-11.638, -27.394, 110.533, -15.672, -82.529, 51.077]
  MoveL 5285 to (507.51, 497.61, 11.7) mm, rotated rx 0 ry 90 rz 0 deg; joints [-11.647, -27.392, 110.516, -15.681, -82.515, 51.083]
  Set speed (120.0 mm/s)
  MoveL 5286 to (509.32, 490.68, 11.7) mm, rotated rx 0 ry 90 rz 0 deg; joints [-10.985, -27.383, 110.465, -15.016, -82.453, 51.017]
  Set speed (30.0 mm/s)
  Call Extruder(0.767)
  MoveL 5287 to (490.68, 509.32, 11.7) mm, rotated rx 0 ry 90 rz 0 deg; joints [-13.056, -27.652, 112.215, -17.051, -83.938, 50.82]
  MoveL 5288 to (490.56, 509.44, 11.7) mm, rotated rx 0 ry 90 rz 0 deg; joints [-13.07, -27.654, 112.226, -17.065, -83.947, 50.819]
  Set speed (120.0 mm/s)
  MoveL 5289 to (497.22, 492.37, 11.7) mm, rotated rx 0 ry 90 rz 0 deg; joints [-11.359, -27.603, 111.874, -15.354, -83.612, 50.743]
  Set speed (1000.0 mm/s)
  MoveL 5290 to (497.29, 492.3, 11.7) mm, rotated rx 0 ry 90 rz 0 deg; joints [-11.351, -27.602, 111.867, -15.346, -83.606, 50.743]
  Set speed (15.0 mm/s)
  Call Extruder(0.119)
  MoveL 5291 to (501.4, 492.3, 11.7) mm, rotated rx 0 ry 90 rz 0 deg; joints [-11.275, -27.528, 111.378, -15.283, -83.203, 50.846]
  Call Extruder(0.010)
  MoveL 5292 to (501.75, 492.3, 11.7) mm, rotated rx 0 ry 90 rz 0 deg; joints [-11.269, -27.521, 111.336, -15.277, -83.169, 50.855]
  Call Extruder(0.007)
  MoveL 5293 to (501.75, 491.95, 11.7) mm, rotated rx 0 ry 90 rz 0 deg; joints [-11.237, -27.523, 111.344, -15.245, -83.175, 50.85]
  Call Extruder(0.035)
  MoveL 5294 to (501.75, 490.75, 11.7) mm, rotated rx 0 ry 90 rz 0 deg; joints [-11.127, -27.527, 111.372, -15.133, -83.195, 50.832]
  Call Extruder(0.010)
  MoveL 5295 to (501.75, 490.4, 11.7) mm, rotated rx 0 ry 90 rz 0 deg; joints [-11.095, -27.528, 111.381, -15.101, -83.201, 50.827]
  Call Extruder(0.007)
  MoveL 5296 to (502.1, 490.4, 11.7) mm, rotated rx 0 ry 90 rz 0 deg; joints [-11.088, -27.522, 111.339, -15.095, -83.166, 50.835]
  Call Extruder(0.218)
  MoveL 5297 to (509.6, 490.4, 11.7) mm, rotated rx 0 ry 90 rz 0 deg; joints [-10.955, -27.379, 110.437, -14.986, -82.43, 51.019]
  Call Extruder(0.189)
  MoveL 5298 to (509.6, 496.91, 11.7) mm, rotated rx 0 ry 90 rz 0 deg; joints [-11.545, -27.353, 110.281, -15.586, -82.323, 51.124]
  Call Extruder(0.056)
  MoveL 5299 to (507.67, 496.91, 11.7) mm, rotated rx 0 ry 90 rz 0 deg; joints [-11.581, -27.391, 110.514, -15.615, -82.512, 51.075]
  Call Extruder(0.062)
  MoveL 5300 to (507.67, 499.05, 11.7) mm, rotated rx 0 ry 90 rz 0 deg; joints [-11.775, -27.383, 110.461, -15.811, -82.475, 51.11]
  Call Extruder(0.010)
  MoveL 5301 to (507.67, 499.4, 11.7) mm, rotated rx 0 ry 90 rz 0 deg; joints [-11.806, -27.381, 110.452, -15.844, -82.469, 51.116]
  Call Extruder(0.007)
  MoveL 5302 to (508.02, 499.4, 11.7) mm, rotated rx 0 ry 90 rz 0 deg; joints [-11.8, -27.374, 110.41, -15.838, -82.435, 51.125]
  Call Extruder(0.046)
  MoveL 5303 to (509.6, 499.4, 11.7) mm, rotated rx 0 ry 90 rz 0 deg; joints [-11.77, -27.343, 110.219, -15.814, -82.281, 51.165]
  Call Extruder(0.010)
  MoveL 5304 to (509.6, 499.75, 11.7) mm, rotated rx 0 ry 90 rz 0 deg; joints [-11.802, -27.342, 110.211, -15.846, -82.275, 51.171]
  Call Extruder(0.046)
  MoveL 5305 to (508.02, 499.74, 11.7) mm, rotated rx 0 ry 90 rz 0 deg; joints [-11.831, -27.373, 110.401, -15.87, -82.429, 51.13]
  Call Extruder(0.010)
  MoveL 5306 to (507.67, 499.74, 11.7) mm, rotated rx 0 ry 90 rz 0 deg; joints [-11.838, -27.38, 110.444, -15.876, -82.463, 51.121]
  Call Extruder(0.007)
  MoveL 5307 to (507.67, 500.09, 11.7) mm, rotated rx 0 ry 90 rz 0 deg; joints [-11.869, -27.378, 110.435, -15.908, -82.457, 51.127]
  Call Extruder(0.062)
  MoveL 5308 to (507.66, 502.22, 11.7) mm, rotated rx 0 ry 90 rz 0 deg; joints [-12.062, -27.37, 110.381, -16.103, -82.42, 51.162]
  Call Extruder(0.056)
  MoveL 5309 to (509.6, 502.22, 11.7) mm, rotated rx 0 ry 90 rz 0 deg; joints [-12.025, -27.331, 110.148, -16.073, -82.232, 51.212]
  Call Extruder(0.215)
  MoveL 5310 to (509.6, 509.6, 11.7) mm, rotated rx 0 ry 90 rz 0 deg; joints [-12.688, -27.299, 109.953, -16.749, -82.1, 51.34]
  Call Extruder(0.559)
  MoveL 5311 to (490.4, 509.6, 11.7) mm, rotated rx 0 ry 90 rz 0 deg; joints [-13.088, -27.656, 112.24, -17.083, -83.959, 50.817]
  MoveL 5312 to (490.4, 490.4, 11.7) mm, rotated rx 0 ry 90 rz 0 deg; joints [-11.303, -27.725, 112.73, -15.277, -84.318, 50.543]
  Call Extruder(0.190)
  MoveL 5313 to (496.94, 490.4, 11.7) mm, rotated rx 0 ry 90 rz 0 deg; joints [-11.182, -27.614, 111.954, -15.174, -83.673, 50.708]
  Call Extruder(0.010)
  MoveL 5314 to (497.3, 490.4, 11.7) mm, rotated rx 0 ry 90 rz 0 deg; joints [-11.176, -27.608, 111.912, -15.168, -83.639, 50.716]
  Call Extruder(0.007)
  MoveL 5315 to (497.29, 490.75, 11.7) mm, rotated rx 0 ry 90 rz 0 deg; joints [-11.208, -27.607, 111.904, -15.201, -83.633, 50.721]
  Call Extruder(0.045)
  MoveL 5316 to (497.29, 492.3, 11.7) mm, rotated rx 0 ry 90 rz 0 deg; joints [-11.351, -27.602, 111.867, -15.346, -83.606, 50.743]
  Set speed (120.0 mm/s)
  MoveL 5317 to (497.69, 492.3, 11.7) mm, rotated rx 0 ry 90 rz 0 deg; joints [-11.344, -27.594, 111.82, -15.34, -83.567, 50.754]
  Set speed (1000.0 mm/s)
  MoveL 5318 to (497.69, 493, 11.7) mm, rotated rx 0 ry 90 rz 0 deg; joints [-11.408, -27.592, 111.803, -15.405, -83.555, 50.764]
  Set speed (1000.0 mm/s)
  MoveL 5319 to (490.68, 490.68, 11.7) mm, rotated rx 0 ry 90 rz 0 deg; joints [-11.324, -27.72, 112.69, -15.299, -84.286, 50.554]
  Set speed (1000.0 mm/s)
  MoveL 5320 to (490.68, 490.68, 11.8) mm, rotated rx 0 ry 90 rz 0 deg; joints [-11.324, -27.73, 112.696, -15.299, -84.28, 50.555]
  Set speed (30.0 mm/s)
  Call Extruder(0.767)
  MoveL 5321 to (509.32, 509.32, 11.8) mm, rotated rx 0 ry 90 rz 0 deg; joints [-12.669, -27.316, 110, -16.728, -82.127, 51.329]
  MoveL 5322 to (509.44, 509.44, 11.8) mm, rotated rx 0 ry 90 rz 0 deg; joints [-12.677, -27.313, 109.981, -16.737, -82.113, 51.334]
  Set speed (120.0 mm/s)
  MoveL 5323 to (507.38, 502.51, 11.8) mm, rotated rx 0 ry 90 rz 0 deg; joints [-12.094, -27.384, 110.412, -16.135, -82.437, 51.161]
  Set speed (30.0 mm/s)
  Call Extruder(0.280)
  MoveL 5324 to (500.58, 509.32, 11.8) mm, rotated rx 0 ry 90 rz 0 deg; joints [-12.847, -27.486, 111.046, -16.875, -82.973, 51.094]
  Set speed (120.0 mm/s)
  MoveL 5325 to (499.42, 509.32, 11.8) mm, rotated rx 0 ry 90 rz 0 deg; joints [-12.872, -27.508, 111.185, -16.895, -83.085, 51.062]
  Set speed (30.0 mm/s)
  Call Extruder(0.360)
  MoveL 5326 to (490.68, 500.58, 11.8) mm, rotated rx 0 ry 90 rz 0 deg; joints [-12.247, -27.696, 112.451, -16.232, -84.101, 50.692]
  Set speed (120.0 mm/s)
  MoveL 5327 to (490.68, 499.42, 11.8) mm, rotated rx 0 ry 90 rz 0 deg; joints [-12.139, -27.7, 112.481, -16.123, -84.123, 50.676]
  Set speed (30.0 mm/s)
  Call Extruder(0.282)
  MoveL 5328 to (497.52, 492.58, 11.8) mm, rotated rx 0 ry 90 rz 0 deg; joints [-11.373, -27.607, 111.839, -15.369, -83.574, 50.755]
  MoveL 5329 to (497.64, 492.45, 11.8) mm, rotated rx 0 ry 90 rz 0 deg; joints [-11.359, -27.605, 111.827, -15.356, -83.564, 50.756]
  Set speed (120.0 mm/s)
  MoveL 5330 to (501.84, 492.33, 11.8) mm, rotated rx 0 ry 90 rz 0 deg; joints [-11.27, -27.53, 111.329, -15.279, -83.154, 50.859]
  Set speed (1000.0 mm/s)
  MoveL 5331 to (502.09, 492.19, 11.8) mm, rotated rx 0 ry 90 rz 0 deg; joints [-11.253, -27.526, 111.302, -15.262, -83.132, 50.863]
  Set speed (30.0 mm/s)
  Call Extruder(0.218)
  MoveL 5332 to (507.39, 497.49, 11.8) mm, rotated rx 0 ry 90 rz 0 deg; joints [-11.638, -27.405, 110.539, -15.672, -82.524, 51.079]
  MoveL 5333 to (507.51, 497.61, 11.8) mm, rotated rx 0 ry 90 rz 0 deg; joints [-11.647, -27.402, 110.521, -15.682, -82.51, 51.084]
  Set speed (120.0 mm/s)
  MoveL 5334 to (509.32, 490.68, 11.8) mm, rotated rx 0 ry 90 rz 0 deg; joints [-10.985, -27.394, 110.47, -15.016, -82.448, 51.018]
  Set speed (30.0 mm/s)
  Call Extruder(0.767)
  MoveL 5335 to (490.68, 509.32, 11.8) mm, rotated rx 0 ry 90 rz 0 deg; joints [-13.056, -27.663, 112.22, -17.051, -83.933, 50.822]
  MoveL 5336 to (490.56, 509.44, 11.8) mm, rotated rx 0 ry 90 rz 0 deg; joints [-13.07, -27.665, 112.231, -17.065, -83.942, 50.821]
  Set speed (120.0 mm/s)
  MoveL 5337 to (497.17, 492.37, 11.8) mm, rotated rx 0 ry 90 rz 0 deg; joints [-11.36, -27.614, 111.886, -15.355, -83.612, 50.743]
  Set speed (1000.0 mm/s)
  MoveL 5338 to (497.24, 492.3, 11.8) mm, rotated rx 0 ry 90 rz 0 deg; joints [-11.352, -27.613, 111.879, -15.347, -83.607, 50.743]
  Set speed (15.0 mm/s)
  Call Extruder(0.123)
  MoveL 5339 to (501.46, 492.3, 11.8) mm, rotated rx 0 ry 90 rz 0 deg; joints [-11.274, -27.537, 111.375, -15.282, -83.192, 50.849]
  Call Extruder(0.010)
  MoveL 5340 to (501.81, 492.3, 11.8) mm, rotated rx 0 ry 90 rz 0 deg; joints [-11.268, -27.531, 111.333, -15.277, -83.158, 50.858]
  Call Extruder(0.007)
  MoveL 5341 to (501.81, 491.95, 11.8) mm, rotated rx 0 ry 90 rz 0 deg; joints [-11.236, -27.532, 111.342, -15.244, -83.163, 50.853]
  Call Extruder(0.035)
  MoveL 5342 to (501.81, 490.75, 11.8) mm, rotated rx 0 ry 90 rz 0 deg; joints [-11.126, -27.536, 111.37, -15.132, -83.184, 50.835]
  Call Extruder(0.010)
  MoveL 5343 to (501.81, 490.4, 11.8) mm, rotated rx 0 ry 90 rz 0 deg; joints [-11.094, -27.538, 111.378, -15.1, -83.189, 50.83]
  Call Extruder(0.007)
  MoveL 5344 to (502.16, 490.4, 11.8) mm, rotated rx 0 ry 90 rz 0 deg; joints [-11.087, -27.531, 111.336, -15.095, -83.155, 50.838]
  Call Extruder(0.216)
  MoveL 5345 to (509.6, 490.4, 11.8) mm, rotated rx 0 ry 90 rz 0 deg; joints [-10.955, -27.389, 110.443, -14.986, -82.425, 51.02]
  Call Extruder(0.188)
  MoveL 5346 to (509.6, 496.85, 11.8) mm, rotated rx 0 ry 90 rz 0 deg; joints [-11.54, -27.364, 110.288, -15.58, -82.319, 51.124]
  Call Extruder(0.056)
  MoveL 5347 to (507.67, 496.85, 11.8) mm, rotated rx 0 ry 90 rz 0 deg; joints [-11.576, -27.402, 110.52, -15.609, -82.507, 51.076]
  Call Extruder(0.062)
  MoveL 5348 to (507.67, 498.99, 11.8) mm, rotated rx 0 ry 90 rz 0 deg; joints [-11.769, -27.393, 110.467, -15.806, -82.471, 51.11]
  Call Extruder(0.010)
  MoveL 5349 to (507.67, 499.34, 11.8) mm, rotated rx 0 ry 90 rz 0 deg; joints [-11.801, -27.392, 110.459, -15.838, -82.465, 51.116]
  Call Extruder(0.007)
  MoveL 5350 to (508.02, 499.34, 11.8) mm, rotated rx 0 ry 90 rz 0 deg; joints [-11.794, -27.385, 110.417, -15.833, -82.431, 51.125]
  Call Extruder(0.046)
  MoveL 5351 to (509.6, 499.34, 11.8) mm, rotated rx 0 ry 90 rz 0 deg; joints [-11.764, -27.354, 110.226, -15.809, -82.277, 51.165]
  Call Extruder(0.014)
  MoveL 5352 to (509.6, 499.8, 11.8) mm, rotated rx 0 ry 90 rz 0 deg; joints [-11.807, -27.352, 110.214, -15.852, -82.269, 51.173]
  Call Extruder(0.046)
  MoveL 5353 to (508.02, 499.8, 11.8) mm, rotated rx 0 ry 90 rz 0 deg; joints [-11.836, -27.383, 110.405, -15.875, -82.423, 51.133]
  Call Extruder(0.010)
  MoveL 5354 to (507.67, 499.8, 11.8) mm, rotated rx 0 ry 90 rz 0 deg; joints [-11.843, -27.39, 110.447, -15.881, -82.457, 51.124]
  Call Extruder(0.007)
  MoveL 5355 to (507.67, 500.15, 11.8) mm, rotated rx 0 ry 90 rz 0 deg; joints [-11.874, -27.389, 110.438, -15.913, -82.451, 51.13]
  Call Extruder(0.062)
  MoveL 5356 to (507.66, 502.28, 11.8) mm, rotated rx 0 ry 90 rz 0 deg; joints [-12.067, -27.38, 110.384, -16.109, -82.414, 51.165]
  Call Extruder(0.056)
  MoveL 5357 to (509.6, 502.28, 11.8) mm, rotated rx 0 ry 90 rz 0 deg; joints [-12.03, -27.341, 110.151, -16.079, -82.226, 51.215]
  Call Extruder(0.213)
  MoveL 5358 to (509.6, 509.6, 11.8) mm, rotated rx 0 ry 90 rz 0 deg; joints [-12.688, -27.309, 109.958, -16.749, -82.095, 51.341]
  Call Extruder(0.559)
  MoveL 5359 to (490.4, 509.6, 11.8) mm, rotated rx 0 ry 90 rz 0 deg; joints [-13.088, -27.667, 112.245, -17.083, -83.954, 50.819]
  MoveL 5360 to (490.4, 490.4, 11.8) mm, rotated rx 0 ry 90 rz 0 deg; joints [-11.303, -27.736, 112.735, -15.277, -84.313, 50.544]
  Call Extruder(0.189)
  MoveL 5361 to (496.89, 490.4, 11.8) mm, rotated rx 0 ry 90 rz 0 deg; joints [-11.183, -27.626, 111.966, -15.175, -83.674, 50.708]
  Call Extruder(0.010)
  MoveL 5362 to (497.24, 490.4, 11.8) mm, rotated rx 0 ry 90 rz 0 deg; joints [-11.177, -27.62, 111.924, -15.169, -83.639, 50.716]
  Call Extruder(0.007)
  MoveL 5363 to (497.24, 490.75, 11.8) mm, rotated rx 0 ry 90 rz 0 deg; joints [-11.209, -27.619, 111.916, -15.202, -83.633, 50.721]
  Call Extruder(0.045)
  MoveL 5364 to (497.24, 492.3, 11.8) mm, rotated rx 0 ry 90 rz 0 deg; joints [-11.352, -27.613, 111.879, -15.347, -83.607, 50.743]
  Set speed (120.0 mm/s)
  MoveL 5365 to (497.64, 492.3, 11.8) mm, rotated rx 0 ry 90 rz 0 deg; joints [-11.345, -27.606, 111.831, -15.341, -83.567, 50.754]
  Set speed (1000.0 mm/s)
  MoveL 5366 to (497.64, 493, 11.8) mm, rotated rx 0 ry 90 rz 0 deg; joints [-11.41, -27.604, 111.815, -15.407, -83.555, 50.764]
  Set speed (1000.0 mm/s)
  MoveL 5367 to (490.68, 490.68, 11.8) mm, rotated rx 0 ry 90 rz 0 deg; joints [-11.324, -27.73, 112.696, -15.299, -84.28, 50.555]
  Set speed (1000.0 mm/s)
  MoveL 5368 to (490.68, 490.68, 11.9) mm, rotated rx 0 ry 90 rz 0 deg; joints [-11.324, -27.741, 112.701, -15.299, -84.275, 50.557]
  Set speed (30.0 mm/s)
  Call Extruder(0.767)
  MoveL 5369 to (509.32, 509.32, 11.9) mm, rotated rx 0 ry 90 rz 0 deg; joints [-12.669, -27.326, 110.005, -16.728, -82.122, 51.33]
  MoveL 5370 to (509.44, 509.44, 11.9) mm, rotated rx 0 ry 90 rz 0 deg; joints [-12.677, -27.323, 109.987, -16.737, -82.108, 51.336]
  Set speed (120.0 mm/s)
  MoveL 5371 to (507.38, 502.51, 11.9) mm, rotated rx 0 ry 90 rz 0 deg; joints [-12.094, -27.395, 110.417, -16.135, -82.432, 51.163]
  Set speed (30.0 mm/s)
  Call Extruder(0.280)
  MoveL 5372 to (500.58, 509.32, 11.9) mm, rotated rx 0 ry 90 rz 0 deg; joints [-12.847, -27.497, 111.052, -16.875, -82.968, 51.095]
  Set speed (120.0 mm/s)
  MoveL 5373 to (499.42, 509.32, 11.9) mm, rotated rx 0 ry 90 rz 0 deg; joints [-12.872, -27.518, 111.19, -16.895, -83.08, 51.064]
  Set speed (30.0 mm/s)
  Call Extruder(0.360)
  MoveL 5374 to (490.68, 500.58, 11.9) mm, rotated rx 0 ry 90 rz 0 deg; joints [-12.247, -27.707, 112.457, -16.232, -84.096, 50.694]
  Set speed (120.0 mm/s)
  MoveL 5375 to (490.68, 499.42, 11.9) mm, rotated rx 0 ry 90 rz 0 deg; joints [-12.139, -27.711, 112.486, -16.123, -84.117, 50.677]
  Set speed (30.0 mm/s)
  Call Extruder(0.282)
  MoveL 5376 to (497.52, 492.58, 11.9) mm, rotated rx 0 ry 90 rz 0 deg; joints [-11.373, -27.618, 111.844, -15.369, -83.569, 50.756]
  MoveL 5377 to (497.64, 492.46, 11.9) mm, rotated rx 0 ry 90 rz 0 deg; joints [-11.359, -27.616, 111.832, -15.356, -83.559, 50.757]
  Set speed (120.0 mm/s)
  MoveL 5378 to (501.9, 492.33, 11.9) mm, rotated rx 0 ry 90 rz 0 deg; joints [-11.269, -27.539, 111.327, -15.278, -83.143, 50.862]
  Set speed (1000.0 mm/s)
  MoveL 5379 to (502.15, 492.26, 11.9) mm, rotated rx 0 ry 90 rz 0 deg; joints [-11.258, -27.535, 111.298, -15.268, -83.12, 50.867]
  Set speed (30.0 mm/s)
  Call Extruder(0.215)
  MoveL 5380 to (507.39, 497.49, 11.9) mm, rotated rx 0 ry 90 rz 0 deg; joints [-11.638, -27.415, 110.544, -15.672, -82.519, 51.08]
  MoveL 5381 to (507.51, 497.61, 11.9) mm, rotated rx 0 ry 90 rz 0 deg; joints [-11.647, -27.413, 110.526, -15.682, -82.505, 51.085]
  Set speed (120.0 mm/s)
  MoveL 5382 to (509.32, 490.68, 11.9) mm, rotated rx 0 ry 90 rz 0 deg; joints [-10.985, -27.404, 110.475, -15.016, -82.443, 51.019]
  Set speed (30.0 mm/s)
  Call Extruder(0.767)
  MoveL 5383 to (490.68, 509.32, 11.9) mm, rotated rx 0 ry 90 rz 0 deg; joints [-13.056, -27.674, 112.225, -17.052, -83.927, 50.824]
  MoveL 5384 to (490.56, 509.44, 11.9) mm, rotated rx 0 ry 90 rz 0 deg; joints [-13.07, -27.675, 112.236, -17.065, -83.937, 50.822]
  Set speed (120.0 mm/s)
  MoveL 5385 to (507.6, 499.35, 11.9) mm, rotated rx 0 ry 90 rz 0 deg; joints [-11.803, -27.404, 110.472, -15.841, -82.466, 51.116]
  Set speed (1000.0 mm/s)
  MoveL 5386 to (507.67, 499.28, 11.9) mm, rotated rx 0 ry 90 rz 0 deg; joints [-11.796, -27.403, 110.465, -15.833, -82.461, 51.117]
  Set speed (15.0 mm/s)
  Call Extruder(0.010)
  MoveL 5387 to (508.02, 499.28, 11.9) mm, rotated rx 0 ry 90 rz 0 deg; joints [-11.789, -27.396, 110.423, -15.828, -82.427, 51.126]
  Call Extruder(0.046)
  MoveL 5388 to (509.6, 499.28, 11.9) mm, rotated rx 0 ry 90 rz 0 deg; joints [-11.759, -27.364, 110.233, -15.804, -82.273, 51.166]
  Call Extruder(0.017)
  MoveL 5389 to (509.6, 499.86, 11.9) mm, rotated rx 0 ry 90 rz 0 deg; joints [-11.812, -27.362, 110.218, -15.857, -82.263, 51.176]
  Call Extruder(0.046)
  MoveL 5390 to (508.02, 499.86, 11.9) mm, rotated rx 0 ry 90 rz 0 deg; joints [-11.841, -27.393, 110.409, -15.881, -82.417, 51.135]
  Call Extruder(0.010)
  MoveL 5391 to (507.67, 499.86, 11.9) mm, rotated rx 0 ry 90 rz 0 deg; joints [-11.848, -27.4, 110.451, -15.886, -82.451, 51.126]
  Call Extruder(0.007)
  MoveL 5392 to (507.67, 500.21, 11.9) mm, rotated rx 0 ry 90 rz 0 deg; joints [-11.88, -27.399, 110.442, -15.919, -82.445, 51.132]
  Call Extruder(0.062)
  MoveL 5393 to (507.67, 502.33, 11.9) mm, rotated rx 0 ry 90 rz 0 deg; joints [-12.072, -27.39, 110.388, -16.114, -82.408, 51.167]
  Call Extruder(0.056)
  MoveL 5394 to (509.6, 502.33, 11.9) mm, rotated rx 0 ry 90 rz 0 deg; joints [-12.035, -27.352, 110.155, -16.084, -82.22, 51.217]
  Call Extruder(0.211)
  MoveL 5395 to (509.6, 509.6, 11.9) mm, rotated rx 0 ry 90 rz 0 deg; joints [-12.688, -27.32, 109.963, -16.749, -82.09, 51.343]
  Call Extruder(0.559)
  MoveL 5396 to (490.4, 509.6, 11.9) mm, rotated rx 0 ry 90 rz 0 deg; joints [-13.088, -27.677, 112.25, -17.083, -83.949, 50.82]
  MoveL 5397 to (490.4, 490.4, 11.9) mm, rotated rx 0 ry 90 rz 0 deg; joints [-11.303, -27.747, 112.74, -15.277, -84.308, 50.546]
  Call Extruder(0.197)
  MoveL 5398 to (497.18, 490.4, 11.9) mm, rotated rx 0 ry 90 rz 0 deg; joints [-11.178, -27.631, 111.936, -15.17, -83.639, 50.716]
  Call Extruder(0.045)
  MoveL 5399 to (497.18, 491.95, 11.9) mm, rotated rx 0 ry 90 rz 0 deg; joints [-11.321, -27.626, 111.899, -15.316, -83.613, 50.738]
  Call Extruder(0.010)
  MoveL 5400 to (497.18, 492.3, 11.9) mm, rotated rx 0 ry 90 rz 0 deg; joints [-11.353, -27.625, 111.891, -15.348, -83.607, 50.744]
  Call Extruder(0.007)
  MoveL 5401 to (497.53, 492.3, 11.9) mm, rotated rx 0 ry 90 rz 0 deg; joints [-11.347, -27.619, 111.849, -15.343, -83.573, 50.752]
  Call Extruder(0.116)
  MoveL 5402 to (501.53, 492.3, 11.9) mm, rotated rx 0 ry 90 rz 0 deg; joints [-11.273, -27.546, 111.373, -15.281, -83.18, 50.852]
  Call Extruder(0.010)
  MoveL 5403 to (501.88, 492.3, 11.9) mm, rotated rx 0 ry 90 rz 0 deg; joints [-11.267, -27.54, 111.331, -15.276, -83.146, 50.861]
  Call Extruder(0.007)
  MoveL 5404 to (501.88, 491.95, 11.9) mm, rotated rx 0 ry 90 rz 0 deg; joints [-11.235, -27.541, 111.339, -15.243, -83.152, 50.856]
  Call Extruder(0.035)
  MoveL 5405 to (501.88, 490.75, 11.9) mm, rotated rx 0 ry 90 rz 0 deg; joints [-11.125, -27.546, 111.367, -15.132, -83.172, 50.838]
  Call Extruder(0.010)
  MoveL 5406 to (501.88, 490.4, 11.9) mm, rotated rx 0 ry 90 rz 0 deg; joints [-11.092, -27.547, 111.376, -15.099, -83.178, 50.833]
  Call Extruder(0.007)
  MoveL 5407 to (502.23, 490.4, 11.9) mm, rotated rx 0 ry 90 rz 0 deg; joints [-11.086, -27.541, 111.334, -15.094, -83.144, 50.841]
  Call Extruder(0.215)
  MoveL 5408 to (509.6, 490.4, 11.9) mm, rotated rx 0 ry 90 rz 0 deg; joints [-10.955, -27.4, 110.448, -14.986, -82.42, 51.022]
  Call Extruder(0.186)
  MoveL 5409 to (509.6, 496.79, 11.9) mm, rotated rx 0 ry 90 rz 0 deg; joints [-11.534, -27.375, 110.294, -15.575, -82.315, 51.125]
  Call Extruder(0.056)
  MoveL 5410 to (507.67, 496.79, 11.9) mm, rotated rx 0 ry 90 rz 0 deg; joints [-11.57, -27.413, 110.527, -15.604, -82.503, 51.076]
  Call Extruder(0.062)
  MoveL 5411 to (507.67, 498.93, 11.9) mm, rotated rx 0 ry 90 rz 0 deg; joints [-11.764, -27.404, 110.474, -15.801, -82.467, 51.111]
  Call Extruder(0.007)
  MoveL 5412 to (507.67, 499.28, 11.9) mm, rotated rx 0 ry 90 rz 0 deg; joints [-11.796, -27.403, 110.465, -15.833, -82.461, 51.117]
  Set speed (120.0 mm/s)
  MoveL 5413 to (508.02, 499.28, 11.9) mm, rotated rx 0 ry 90 rz 0 deg; joints [-11.789, -27.396, 110.423, -15.828, -82.427, 51.126]
  Set speed (1000.0 mm/s)
  MoveL 5414 to (508.07, 499.28, 11.9) mm, rotated rx 0 ry 90 rz 0 deg; joints [-11.788, -27.395, 110.417, -15.827, -82.422, 51.127]
  Set speed (1000.0 mm/s)
  MoveL 5415 to (508.07, 499.38, 11.9) mm, rotated rx 0 ry 90 rz 0 deg; joints [-11.797, -27.394, 110.415, -15.836, -82.42, 51.129]
  Set speed (1000.0 mm/s)
  MoveL 5416 to (490.68, 490.68, 11.9) mm, rotated rx 0 ry 90 rz 0 deg; joints [-11.324, -27.741, 112.701, -15.299, -84.275, 50.557]
  Set speed (1000.0 mm/s)
  MoveL 5417 to (490.68, 490.68, 12) mm, rotated rx 0 ry 90 rz 0 deg; joints [-11.324, -27.752, 112.706, -15.299, -84.27, 50.558]
  Set speed (30.0 mm/s)
  Call Extruder(0.767)
  MoveL 5418 to (509.32, 509.32, 12) mm, rotated rx 0 ry 90 rz 0 deg; joints [-12.669, -27.337, 110.01, -16.728, -82.117, 51.332]
  MoveL 5419 to (509.44, 509.44, 12) mm, rotated rx 0 ry 90 rz 0 deg; joints [-12.677, -27.334, 109.992, -16.738, -82.103, 51.337]
  Set speed (120.0 mm/s)
  MoveL 5420 to (507.39, 502.51, 12) mm, rotated rx 0 ry 90 rz 0 deg; joints [-12.094, -27.405, 110.422, -16.135, -82.427, 51.164]
  Set speed (30.0 mm/s)
  Call Extruder(0.280)
  MoveL 5421 to (500.58, 509.32, 12) mm, rotated rx 0 ry 90 rz 0 deg; joints [-12.847, -27.507, 111.057, -16.875, -82.963, 51.097]
  Set speed (120.0 mm/s)
  MoveL 5422 to (499.42, 509.32, 12) mm, rotated rx 0 ry 90 rz 0 deg; joints [-12.872, -27.529, 111.195, -16.895, -83.075, 51.066]
  Set speed (30.0 mm/s)
  Call Extruder(0.360)
  MoveL 5423 to (490.68, 500.58, 12) mm, rotated rx 0 ry 90 rz 0 deg; joints [-12.247, -27.717, 112.462, -16.232, -84.091, 50.695]
  Set speed (120.0 mm/s)
  MoveL 5424 to (490.68, 499.42, 12) mm, rotated rx 0 ry 90 rz 0 deg; joints [-12.139, -27.722, 112.492, -16.123, -84.112, 50.679]
  Set speed (30.0 mm/s)
  Call Extruder(0.282)
  MoveL 5425 to (497.52, 492.58, 12) mm, rotated rx 0 ry 90 rz 0 deg; joints [-11.373, -27.628, 111.849, -15.369, -83.564, 50.757]
  MoveL 5426 to (497.64, 492.46, 12) mm, rotated rx 0 ry 90 rz 0 deg; joints [-11.359, -27.627, 111.837, -15.356, -83.554, 50.759]
  Set speed (120.0 mm/s)
  MoveL 5427 to (502.22, 492.32, 12) mm, rotated rx 0 ry 90 rz 0 deg; joints [-11.262, -27.544, 111.294, -15.273, -83.107, 50.871]
  Set speed (30.0 mm/s)
  Call Extruder(0.213)
  MoveL 5428 to (507.39, 497.49, 12) mm, rotated rx 0 ry 90 rz 0 deg; joints [-11.638, -27.426, 110.549, -15.673, -82.514, 51.082]
  MoveL 5429 to (507.51, 497.61, 12) mm, rotated rx 0 ry 90 rz 0 deg; joints [-11.647, -27.423, 110.531, -15.682, -82.5, 51.087]
  Set speed (120.0 mm/s)
  MoveL 5430 to (509.32, 490.68, 12) mm, rotated rx 0 ry 90 rz 0 deg; joints [-10.985, -27.415, 110.48, -15.016, -82.438, 51.021]
  Set speed (30.0 mm/s)
  Call Extruder(0.767)
  MoveL 5431 to (490.68, 509.32, 12) mm, rotated rx 0 ry 90 rz 0 deg; joints [-13.056, -27.684, 112.23, -17.052, -83.922, 50.825]
  MoveL 5432 to (490.56, 509.44, 12) mm, rotated rx 0 ry 90 rz 0 deg; joints [-13.07, -27.686, 112.242, -17.066, -83.932, 50.824]
  Set speed (120.0 mm/s)
  MoveL 5433 to (507.6, 499.29, 12) mm, rotated rx 0 ry 90 rz 0 deg; joints [-11.798, -27.415, 110.479, -15.836, -82.462, 51.117]
  Set speed (1000.0 mm/s)
  MoveL 5434 to (507.67, 499.22, 12) mm, rotated rx 0 ry 90 rz 0 deg; joints [-11.79, -27.413, 110.472, -15.828, -82.457, 51.117]
  Set speed (15.0 mm/s)
  Call Extruder(0.010)
  MoveL 5435 to (508.02, 499.22, 12) mm, rotated rx 0 ry 90 rz 0 deg; joints [-11.784, -27.407, 110.43, -15.823, -82.423, 51.126]
  Call Extruder(0.046)
  MoveL 5436 to (509.6, 499.22, 12) mm, rotated rx 0 ry 90 rz 0 deg; joints [-11.754, -27.375, 110.239, -15.798, -82.269, 51.166]
  Call Extruder(0.020)
  MoveL 5437 to (509.6, 499.92, 12) mm, rotated rx 0 ry 90 rz 0 deg; joints [-11.817, -27.372, 110.222, -15.862, -82.257, 51.178]
  Call Extruder(0.046)
  MoveL 5438 to (508.02, 499.91, 12) mm, rotated rx 0 ry 90 rz 0 deg; joints [-11.846, -27.404, 110.413, -15.886, -82.411, 51.137]
  Call Extruder(0.010)
  MoveL 5439 to (507.67, 499.91, 12) mm, rotated rx 0 ry 90 rz 0 deg; joints [-11.853, -27.411, 110.455, -15.892, -82.445, 51.129]
  Call Extruder(0.007)
  MoveL 5440 to (507.67, 500.26, 12) mm, rotated rx 0 ry 90 rz 0 deg; joints [-11.884, -27.409, 110.446, -15.924, -82.439, 51.134]
  Call Extruder(0.062)
  MoveL 5441 to (507.67, 502.39, 12) mm, rotated rx 0 ry 90 rz 0 deg; joints [-12.077, -27.4, 110.392, -16.119, -82.402, 51.17]
  Call Extruder(0.056)
  MoveL 5442 to (509.6, 502.39, 12) mm, rotated rx 0 ry 90 rz 0 deg; joints [-12.04, -27.362, 110.159, -16.09, -82.214, 51.22]
  Call Extruder(0.210)
  MoveL 5443 to (509.6, 509.6, 12) mm, rotated rx 0 ry 90 rz 0 deg; joints [-12.688, -27.33, 109.968, -16.749, -82.085, 51.344]
  Call Extruder(0.559)
  MoveL 5444 to (490.4, 509.6, 12) mm, rotated rx 0 ry 90 rz 0 deg; joints [-13.088, -27.688, 112.256, -17.083, -83.944, 50.822]
  MoveL 5445 to (490.4, 490.4, 12) mm, rotated rx 0 ry 90 rz 0 deg; joints [-11.303, -27.757, 112.746, -15.278, -84.302, 50.547]
  Call Extruder(0.196)
  MoveL 5446 to (497.13, 490.4, 12) mm, rotated rx 0 ry 90 rz 0 deg; joints [-11.179, -27.643, 111.948, -15.171, -83.64, 50.716]
  Call Extruder(0.045)
  MoveL 5447 to (497.13, 491.95, 12) mm, rotated rx 0 ry 90 rz 0 deg; joints [-11.322, -27.638, 111.911, -15.317, -83.613, 50.739]
  Call Extruder(0.010)
  MoveL 5448 to (497.13, 492.3, 12) mm, rotated rx 0 ry 90 rz 0 deg; joints [-11.354, -27.636, 111.903, -15.349, -83.607, 50.744]
  Call Extruder(0.007)
  MoveL 5449 to (497.48, 492.3, 12) mm, rotated rx 0 ry 90 rz 0 deg; joints [-11.348, -27.63, 111.861, -15.344, -83.573, 50.752]
  Call Extruder(0.120)
  MoveL 5450 to (501.59, 492.3, 12) mm, rotated rx 0 ry 90 rz 0 deg; joints [-11.272, -27.556, 111.37, -15.28, -83.169, 50.855]
  Call Extruder(0.010)
  MoveL 5451 to (501.94, 492.3, 12) mm, rotated rx 0 ry 90 rz 0 deg; joints [-11.266, -27.549, 111.328, -15.275, -83.135, 50.864]
  Call Extruder(0.007)
  MoveL 5452 to (501.94, 491.95, 12) mm, rotated rx 0 ry 90 rz 0 deg; joints [-11.233, -27.551, 111.337, -15.242, -83.14, 50.859]
  Call Extruder(0.035)
  MoveL 5453 to (501.94, 490.75, 12) mm, rotated rx 0 ry 90 rz 0 deg; joints [-11.123, -27.555, 111.365, -15.131, -83.161, 50.841]
  Call Extruder(0.010)
  MoveL 5454 to (501.94, 490.4, 12) mm, rotated rx 0 ry 90 rz 0 deg; joints [-11.091, -27.556, 111.373, -15.098, -83.167, 50.836]
  Call Extruder(0.007)
  MoveL 5455 to (502.29, 490.4, 12) mm, rotated rx 0 ry 90 rz 0 deg; joints [-11.085, -27.55, 111.331, -15.093, -83.132, 50.844]
  Call Extruder(0.213)
  MoveL 5456 to (509.6, 490.4, 12) mm, rotated rx 0 ry 90 rz 0 deg; joints [-10.955, -27.41, 110.453, -14.986, -82.415, 51.023]
  Call Extruder(0.184)
  MoveL 5457 to (509.6, 496.73, 12) mm, rotated rx 0 ry 90 rz 0 deg; joints [-11.529, -27.385, 110.301, -15.57, -82.311, 51.125]
  Call Extruder(0.056)
  MoveL 5458 to (507.67, 496.73, 12) mm, rotated rx 0 ry 90 rz 0 deg; joints [-11.565, -27.424, 110.534, -15.599, -82.499, 51.077]
  Call Extruder(0.072)
  MoveL 5459 to (507.67, 499.22, 12) mm, rotated rx 0 ry 90 rz 0 deg; joints [-11.79, -27.413, 110.472, -15.828, -82.457, 51.117]
  Set speed (120.0 mm/s)
  MoveL 5460 to (508.02, 499.22, 12) mm, rotated rx 0 ry 90 rz 0 deg; joints [-11.784, -27.407, 110.43, -15.823, -82.423, 51.126]
  Set speed (1000.0 mm/s)
  MoveL 5461 to (508.07, 499.22, 12) mm, rotated rx 0 ry 90 rz 0 deg; joints [-11.783, -27.406, 110.424, -15.822, -82.418, 51.127]
  Set speed (1000.0 mm/s)
  MoveL 5462 to (508.07, 499.32, 12) mm, rotated rx 0 ry 90 rz 0 deg; joints [-11.792, -27.405, 110.421, -15.831, -82.416, 51.129]
  Set speed (1000.0 mm/s)
  MoveL 5463 to (490.68, 490.68, 12) mm, rotated rx 0 ry 90 rz 0 deg; joints [-11.324, -27.752, 112.706, -15.299, -84.27, 50.558]
  Set speed (1000.0 mm/s)
  MoveL 5464 to (490.68, 490.68, 12.1) mm, rotated rx 0 ry 90 rz 0 deg; joints [-11.324, -27.762, 112.711, -15.3, -84.265, 50.559]
  Set speed (30.0 mm/s)
  Call Extruder(0.767)
  MoveL 5465 to (509.32, 509.32, 12.1) mm, rotated rx 0 ry 90 rz 0 deg; joints [-12.669, -27.347, 110.015, -16.729, -82.112, 51.333]
  MoveL 5466 to (509.44, 509.44, 12.1) mm, rotated rx 0 ry 90 rz 0 deg; joints [-12.677, -27.344, 109.997, -16.738, -82.098, 51.339]
  Set speed (120.0 mm/s)
  MoveL 5467 to (507.38, 502.51, 12.1) mm, rotated rx 0 ry 90 rz 0 deg; joints [-12.094, -27.416, 110.427, -16.136, -82.422, 51.166]
  Set speed (30.0 mm/s)
  Call Extruder(0.280)
  MoveL 5468 to (500.58, 509.32, 12.1) mm, rotated rx 0 ry 90 rz 0 deg; joints [-12.847, -27.518, 111.062, -16.876, -82.958, 51.099]
  Set speed (120.0 mm/s)
  MoveL 5469 to (499.42, 509.32, 12.1) mm, rotated rx 0 ry 90 rz 0 deg; joints [-12.872, -27.539, 111.2, -16.896, -83.07, 51.067]
  Set speed (30.0 mm/s)
  Call Extruder(0.360)
  MoveL 5470 to (490.68, 500.58, 12.1) mm, rotated rx 0 ry 90 rz 0 deg; joints [-12.247, -27.728, 112.467, -16.233, -84.085, 50.697]
  Set speed (120.0 mm/s)
  MoveL 5471 to (490.68, 499.42, 12.1) mm, rotated rx 0 ry 90 rz 0 deg; joints [-12.139, -27.732, 112.497, -16.124, -84.107, 50.68]
  Set speed (30.0 mm/s)
  Call Extruder(0.282)
  MoveL 5472 to (497.52, 492.58, 12.1) mm, rotated rx 0 ry 90 rz 0 deg; joints [-11.373, -27.639, 111.854, -15.37, -83.559, 50.759]
  MoveL 5473 to (497.64, 492.46, 12.1) mm, rotated rx 0 ry 90 rz 0 deg; joints [-11.359, -27.637, 111.843, -15.356, -83.549, 50.76]
  Set speed (120.0 mm/s)
  MoveL 5474 to (502.28, 492.38, 12.1) mm, rotated rx 0 ry 90 rz 0 deg; joints [-11.267, -27.553, 111.29, -15.278, -83.094, 50.875]
  Set speed (30.0 mm/s)
  Call Extruder(0.210)
  MoveL 5475 to (507.39, 497.49, 12.1) mm, rotated rx 0 ry 90 rz 0 deg; joints [-11.638, -27.436, 110.554, -15.673, -82.509, 51.083]
  MoveL 5476 to (507.51, 497.61, 12.1) mm, rotated rx 0 ry 90 rz 0 deg; joints [-11.647, -27.434, 110.536, -15.682, -82.495, 51.088]
  Set speed (120.0 mm/s)
  MoveL 5477 to (509.32, 490.68, 12.1) mm, rotated rx 0 ry 90 rz 0 deg; joints [-10.985, -27.425, 110.485, -15.016, -82.432, 51.022]
  Set speed (30.0 mm/s)
  Call Extruder(0.767)
  MoveL 5478 to (490.68, 509.32, 12.1) mm, rotated rx 0 ry 90 rz 0 deg; joints [-13.056, -27.695, 112.236, -17.052, -83.917, 50.827]
  MoveL 5479 to (490.56, 509.44, 12.1) mm, rotated rx 0 ry 90 rz 0 deg; joints [-13.07, -27.697, 112.247, -17.066, -83.927, 50.825]
  Set speed (120.0 mm/s)
  MoveL 5480 to (502.07, 492.37, 12.1) mm, rotated rx 0 ry 90 rz 0 deg; joints [-11.27, -27.557, 111.316, -15.28, -83.115, 50.87]
  Set speed (1000.0 mm/s)
  MoveL 5481 to (502.01, 492.3, 12.1) mm, rotated rx 0 ry 90 rz 0 deg; joints [-11.264, -27.559, 111.326, -15.274, -83.123, 50.867]
  Set speed (15.0 mm/s)
  Call Extruder(0.010)
  MoveL 5482 to (502.01, 491.95, 12.1) mm, rotated rx 0 ry 90 rz 0 deg; joints [-11.232, -27.56, 111.334, -15.242, -83.129, 50.862]
  Call Extruder(0.035)
  MoveL 5483 to (502, 490.75, 12.1) mm, rotated rx 0 ry 90 rz 0 deg; joints [-11.122, -27.564, 111.363, -15.13, -83.149, 50.844]
  Call Extruder(0.010)
  MoveL 5484 to (502, 490.4, 12.1) mm, rotated rx 0 ry 90 rz 0 deg; joints [-11.09, -27.566, 111.371, -15.097, -83.155, 50.839]
  Call Extruder(0.007)
  MoveL 5485 to (502.35, 490.4, 12.1) mm, rotated rx 0 ry 90 rz 0 deg; joints [-11.084, -27.559, 111.329, -15.092, -83.121, 50.847]
  Call Extruder(0.211)
  MoveL 5486 to (509.6, 490.4, 12.1) mm, rotated rx 0 ry 90 rz 0 deg; joints [-10.955, -27.421, 110.458, -14.987, -82.409, 51.025]
  Call Extruder(0.183)
  MoveL 5487 to (509.6, 496.67, 12.1) mm, rotated rx 0 ry 90 rz 0 deg; joints [-11.523, -27.396, 110.308, -15.564, -82.307, 51.126]
  Call Extruder(0.056)
  MoveL 5488 to (507.67, 496.67, 12.1) mm, rotated rx 0 ry 90 rz 0 deg; joints [-11.559, -27.434, 110.54, -15.594, -82.495, 51.077]
  Call Extruder(0.062)
  MoveL 5489 to (507.67, 498.81, 12.1) mm, rotated rx 0 ry 90 rz 0 deg; joints [-11.753, -27.426, 110.487, -15.791, -82.459, 51.112]
  Call Extruder(0.010)
  MoveL 5490 to (507.67, 499.16, 12.1) mm, rotated rx 0 ry 90 rz 0 deg; joints [-11.785, -27.424, 110.478, -15.823, -82.453, 51.118]
  Call Extruder(0.007)
  MoveL 5491 to (508.02, 499.16, 12.1) mm, rotated rx 0 ry 90 rz 0 deg; joints [-11.778, -27.417, 110.436, -15.818, -82.419, 51.127]
  Call Extruder(0.036)
  MoveL 5492 to (509.25, 499.16, 12.1) mm, rotated rx 0 ry 90 rz 0 deg; joints [-11.755, -27.393, 110.288, -15.799, -82.299, 51.158]
  Call Extruder(0.010)
  MoveL 5493 to (509.6, 499.16, 12.1) mm, rotated rx 0 ry 90 rz 0 deg; joints [-11.749, -27.386, 110.246, -15.793, -82.264, 51.167]
  Call Extruder(0.007)
  MoveL 5494 to (509.6, 499.51, 12.1) mm, rotated rx 0 ry 90 rz 0 deg; joints [-11.78, -27.384, 110.237, -15.825, -82.258, 51.173]
  Call Extruder(0.003)
  MoveL 5495 to (509.6, 499.62, 12.1) mm, rotated rx 0 ry 90 rz 0 deg; joints [-11.79, -27.384, 110.234, -15.835, -82.257, 51.174]
  Call Extruder(0.010)
  MoveL 5496 to (509.6, 499.97, 12.1) mm, rotated rx 0 ry 90 rz 0 deg; joints [-11.822, -27.383, 110.226, -15.867, -82.251, 51.18]
  Call Extruder(0.007)
  MoveL 5497 to (509.25, 499.97, 12.1) mm, rotated rx 0 ry 90 rz 0 deg; joints [-11.828, -27.39, 110.268, -15.873, -82.285, 51.171]
  Call Extruder(0.036)
  MoveL 5498 to (508.02, 499.97, 12.1) mm, rotated rx 0 ry 90 rz 0 deg; joints [-11.851, -27.414, 110.416, -15.892, -82.405, 51.14]
  Call Extruder(0.010)
  MoveL 5499 to (507.67, 499.97, 12.1) mm, rotated rx 0 ry 90 rz 0 deg; joints [-11.858, -27.421, 110.458, -15.897, -82.439, 51.131]
  Call Extruder(0.007)
  MoveL 5500 to (507.67, 500.32, 12.1) mm, rotated rx 0 ry 90 rz 0 deg; joints [-11.89, -27.419, 110.45, -15.929, -82.433, 51.137]
  Call Extruder(0.062)
  MoveL 5501 to (507.67, 502.45, 12.1) mm, rotated rx 0 ry 90 rz 0 deg; joints [-12.082, -27.411, 110.395, -16.125, -82.396, 51.172]
  Call Extruder(0.056)
  MoveL 5502 to (509.6, 502.45, 12.1) mm, rotated rx 0 ry 90 rz 0 deg; joints [-12.045, -27.372, 110.162, -16.095, -82.208, 51.222]
  Call Extruder(0.208)
  MoveL 5503 to (509.6, 509.6, 12.1) mm, rotated rx 0 ry 90 rz 0 deg; joints [-12.688, -27.34, 109.974, -16.75, -82.08, 51.346]
  Call Extruder(0.559)
  MoveL 5504 to (490.4, 509.6, 12.1) mm, rotated rx 0 ry 90 rz 0 deg; joints [-13.088, -27.699, 112.261, -17.083, -83.939, 50.823]
  MoveL 5505 to (490.4, 490.4, 12.1) mm, rotated rx 0 ry 90 rz 0 deg; joints [-11.303, -27.768, 112.751, -15.278, -84.297, 50.549]
  Call Extruder(0.184)
  MoveL 5506 to (496.72, 490.4, 12.1) mm, rotated rx 0 ry 90 rz 0 deg; joints [-11.186, -27.661, 112.001, -15.178, -83.674, 50.708]
  Call Extruder(0.010)
  MoveL 5507 to (497.07, 490.4, 12.1) mm, rotated rx 0 ry 90 rz 0 deg; joints [-11.18, -27.655, 111.96, -15.172, -83.64, 50.716]
  Call Extruder(0.007)
  MoveL 5508 to (497.07, 490.75, 12.1) mm, rotated rx 0 ry 90 rz 0 deg; joints [-11.212, -27.653, 111.951, -15.205, -83.634, 50.721]
  Call Extruder(0.035)
  MoveL 5509 to (497.07, 491.95, 12.1) mm, rotated rx 0 ry 90 rz 0 deg; joints [-11.323, -27.649, 111.923, -15.318, -83.614, 50.739]
  Call Extruder(0.010)
  MoveL 5510 to (497.07, 492.3, 12.1) mm, rotated rx 0 ry 90 rz 0 deg; joints [-11.356, -27.648, 111.915, -15.351, -83.608, 50.744]
  Call Extruder(0.007)
  MoveL 5511 to (497.42, 492.3, 12.1) mm, rotated rx 0 ry 90 rz 0 deg; joints [-11.349, -27.642, 111.873, -15.345, -83.573, 50.752]
  Call Extruder(0.061)
  MoveL 5512 to (499.53, 492.3, 12.1) mm, rotated rx 0 ry 90 rz 0 deg; joints [-11.31, -27.604, 111.621, -15.312, -83.366, 50.805]
  Call Extruder(0.055)
  MoveL 5513 to (499.53, 490.4, 12.1) mm, rotated rx 0 ry 90 rz 0 deg; joints [-11.135, -27.611, 111.666, -15.135, -83.398, 50.778]
  Call Extruder(0.002)
  MoveL 5514 to (499.59, 490.4, 12.1) mm, rotated rx 0 ry 90 rz 0 deg; joints [-11.134, -27.61, 111.66, -15.134, -83.393, 50.779]
  Call Extruder(0.004)
  MoveL 5515 to (499.59, 492.3, 12.1) mm, rotated rx 0 ry 90 rz 0 deg; joints [-11.309, -27.603, 111.615, -15.311, -83.36, 50.807]
  Call Extruder(0.060)
  MoveL 5516 to (501.65, 492.3, 12.1) mm, rotated rx 0 ry 90 rz 0 deg; joints [-11.271, -27.565, 111.368, -15.28, -83.157, 50.858]
  Call Extruder(0.007)
  MoveL 5517 to (502.01, 492.3, 12.1) mm, rotated rx 0 ry 90 rz 0 deg; joints [-11.264, -27.559, 111.326, -15.274, -83.123, 50.867]
  Set speed (120.0 mm/s)
  MoveL 5518 to (502.01, 491.95, 12.1) mm, rotated rx 0 ry 90 rz 0 deg; joints [-11.232, -27.56, 111.334, -15.242, -83.129, 50.862]
  Set speed (1000.0 mm/s)
  MoveL 5519 to (502.01, 491.9, 12.1) mm, rotated rx 0 ry 90 rz 0 deg; joints [-11.228, -27.56, 111.335, -15.237, -83.13, 50.861]
  Set speed (1000.0 mm/s)
  MoveL 5520 to (502.11, 491.9, 12.1) mm, rotated rx 0 ry 90 rz 0 deg; joints [-11.226, -27.558, 111.323, -15.235, -83.12, 50.864]
  Set speed (1000.0 mm/s)
  MoveL 5521 to (507.41, 499.49, 12.1) mm, rotated rx 0 ry 90 rz 0 deg; joints [-11.82, -27.428, 110.501, -15.857, -82.472, 51.117]
  Set speed (1000.0 mm/s)
  MoveL 5522 to (507.48, 499.56, 12.1) mm, rotated rx 0 ry 90 rz 0 deg; joints [-11.825, -27.426, 110.491, -15.863, -82.464, 51.12]
  Set speed (15.0 mm/s)
  Call Extruder(0.004)
  MoveL 5523 to (507.98, 499.56, 12.1) mm, rotated rx 0 ry 90 rz 0 deg; joints [-11.816, -27.416, 110.431, -15.855, -82.415, 51.132]
  Call Extruder(0.008)
  MoveL 5524 to (508.97, 499.57, 12.1) mm, rotated rx 0 ry 90 rz 0 deg; joints [-11.797, -27.397, 110.312, -15.84, -82.319, 51.158]
  Set speed (120.0 mm/s)
  MoveL 5525 to (509.04, 499.86, 12.1) mm, rotated rx 0 ry 90 rz 0 deg; joints [-11.822, -27.394, 110.296, -15.866, -82.307, 51.164]
  Set speed (1000.0 mm/s)
  MoveL 5526 to (490.68, 490.68, 12.1) mm, rotated rx 0 ry 90 rz 0 deg; joints [-11.324, -27.762, 112.711, -15.3, -84.265, 50.559]
  Set speed (1000.0 mm/s)
  MoveL 5527 to (490.68, 490.68, 12.2) mm, rotated rx 0 ry 90 rz 0 deg; joints [-11.324, -27.773, 112.716, -15.3, -84.259, 50.561]
  Set speed (30.0 mm/s)
  Call Extruder(0.767)
  MoveL 5528 to (509.32, 509.32, 12.2) mm, rotated rx 0 ry 90 rz 0 deg; joints [-12.669, -27.358, 110.02, -16.729, -82.107, 51.335]
  MoveL 5529 to (509.44, 509.44, 12.2) mm, rotated rx 0 ry 90 rz 0 deg; joints [-12.677, -27.355, 110.002, -16.738, -82.093, 51.34]
  Set speed (120.0 mm/s)
  MoveL 5530 to (507.38, 502.51, 12.2) mm, rotated rx 0 ry 90 rz 0 deg; joints [-12.094, -27.426, 110.432, -16.136, -82.417, 51.167]
  Set speed (30.0 mm/s)
  Call Extruder(0.280)
  MoveL 5531 to (500.58, 509.32, 12.2) mm, rotated rx 0 ry 90 rz 0 deg; joints [-12.847, -27.528, 111.067, -16.876, -82.953, 51.1]
  Set speed (120.0 mm/s)
  MoveL 5532 to (499.42, 509.32, 12.2) mm, rotated rx 0 ry 90 rz 0 deg; joints [-12.872, -27.55, 111.205, -16.896, -83.065, 51.069]
  Set speed (30.0 mm/s)
  Call Extruder(0.360)
  MoveL 5533 to (490.68, 500.58, 12.2) mm, rotated rx 0 ry 90 rz 0 deg; joints [-12.247, -27.739, 112.472, -16.233, -84.08, 50.698]
  Set speed (120.0 mm/s)
  MoveL 5534 to (490.68, 499.42, 12.2) mm, rotated rx 0 ry 90 rz 0 deg; joints [-12.139, -27.743, 112.502, -16.124, -84.102, 50.682]
  Set speed (30.0 mm/s)
  Call Extruder(0.282)
  MoveL 5535 to (497.52, 492.58, 12.2) mm, rotated rx 0 ry 90 rz 0 deg; joints [-11.373, -27.65, 111.86, -15.37, -83.553, 50.76]
  MoveL 5536 to (497.64, 492.46, 12.2) mm, rotated rx 0 ry 90 rz 0 deg; joints [-11.359, -27.648, 111.848, -15.356, -83.544, 50.762]
  Set speed (120.0 mm/s)
  MoveL 5537 to (502.35, 492.45, 12.2) mm, rotated rx 0 ry 90 rz 0 deg; joints [-11.272, -27.562, 111.286, -15.283, -83.082, 50.879]
  Set speed (30.0 mm/s)
  Call Extruder(0.207)
  MoveL 5538 to (507.39, 497.49, 12.2) mm, rotated rx 0 ry 90 rz 0 deg; joints [-11.639, -27.447, 110.559, -15.673, -82.503, 51.085]
  MoveL 5539 to (507.51, 497.61, 12.2) mm, rotated rx 0 ry 90 rz 0 deg; joints [-11.647, -27.444, 110.541, -15.683, -82.489, 51.09]
  Set speed (120.0 mm/s)
  MoveL 5540 to (509.32, 490.68, 12.2) mm, rotated rx 0 ry 90 rz 0 deg; joints [-10.985, -27.436, 110.491, -15.016, -82.427, 51.024]
  Set speed (30.0 mm/s)
  Call Extruder(0.767)
  MoveL 5541 to (490.68, 509.32, 12.2) mm, rotated rx 0 ry 90 rz 0 deg; joints [-13.056, -27.706, 112.241, -17.052, -83.912, 50.828]
  MoveL 5542 to (490.56, 509.44, 12.2) mm, rotated rx 0 ry 90 rz 0 deg; joints [-13.07, -27.707, 112.252, -17.066, -83.921, 50.827]
  Set speed (120.0 mm/s)
  MoveL 5543 to (496.94, 492.37, 12.2) mm, rotated rx 0 ry 90 rz 0 deg; joints [-11.364, -27.661, 111.933, -15.359, -83.614, 50.743]
  Set speed (1000.0 mm/s)
  MoveL 5544 to (497.01, 492.3, 12.2) mm, rotated rx 0 ry 90 rz 0 deg; joints [-11.357, -27.66, 111.927, -15.352, -83.608, 50.744]
  Set speed (15.0 mm/s)
  Call Extruder(0.072)
  MoveL 5545 to (499.47, 492.3, 12.2) mm, rotated rx 0 ry 90 rz 0 deg; joints [-11.311, -27.616, 111.633, -15.313, -83.366, 50.805]
  Call Extruder(0.055)
  MoveL 5546 to (499.47, 490.4, 12.2) mm, rotated rx 0 ry 90 rz 0 deg; joints [-11.136, -27.622, 111.678, -15.136, -83.398, 50.778]
  Call Extruder(0.005)
  MoveL 5547 to (499.65, 490.4, 12.2) mm, rotated rx 0 ry 90 rz 0 deg; joints [-11.133, -27.619, 111.657, -15.133, -83.381, 50.782]
  Call Extruder(0.014)
  MoveL 5548 to (499.65, 492.3, 12.2) mm, rotated rx 0 ry 90 rz 0 deg; joints [-11.308, -27.612, 111.612, -15.311, -83.349, 50.81]
  Call Extruder(0.060)
  MoveL 5549 to (501.72, 492.3, 12.2) mm, rotated rx 0 ry 90 rz 0 deg; joints [-11.27, -27.575, 111.365, -15.279, -83.146, 50.862]
  Call Extruder(0.010)
  MoveL 5550 to (502.07, 492.3, 12.2) mm, rotated rx 0 ry 90 rz 0 deg; joints [-11.263, -27.568, 111.323, -15.273, -83.112, 50.87]
  Call Extruder(0.007)
  MoveL 5551 to (502.07, 491.95, 12.2) mm, rotated rx 0 ry 90 rz 0 deg; joints [-11.231, -27.569, 111.332, -15.241, -83.118, 50.865]
  Call Extruder(0.035)
  MoveL 5552 to (502.07, 490.75, 12.2) mm, rotated rx 0 ry 90 rz 0 deg; joints [-11.121, -27.574, 111.36, -15.129, -83.138, 50.847]
  Call Extruder(0.010)
  MoveL 5553 to (502.07, 490.4, 12.2) mm, rotated rx 0 ry 90 rz 0 deg; joints [-11.089, -27.575, 111.368, -15.097, -83.144, 50.842]
  Call Extruder(0.007)
  MoveL 5554 to (502.42, 490.4, 12.2) mm, rotated rx 0 ry 90 rz 0 deg; joints [-11.083, -27.569, 111.326, -15.091, -83.109, 50.85]
  Call Extruder(0.209)
  MoveL 5555 to (509.6, 490.4, 12.2) mm, rotated rx 0 ry 90 rz 0 deg; joints [-10.955, -27.431, 110.463, -14.987, -82.404, 51.026]
  Call Extruder(0.181)
  MoveL 5556 to (509.6, 496.61, 12.2) mm, rotated rx 0 ry 90 rz 0 deg; joints [-11.518, -27.407, 110.314, -15.559, -82.302, 51.126]
  Call Extruder(0.056)
  MoveL 5557 to (507.67, 496.61, 12.2) mm, rotated rx 0 ry 90 rz 0 deg; joints [-11.554, -27.445, 110.547, -15.588, -82.491, 51.078]
  Call Extruder(0.072)
  MoveL 5558 to (507.67, 499.1, 12.2) mm, rotated rx 0 ry 90 rz 0 deg; joints [-11.78, -27.435, 110.485, -15.818, -82.448, 51.118]
  Call Extruder(0.056)
  MoveL 5559 to (509.6, 499.1, 12.2) mm, rotated rx 0 ry 90 rz 0 deg; joints [-11.743, -27.397, 110.252, -15.788, -82.26, 51.167]
  Call Extruder(0.017)
  MoveL 5560 to (509.6, 499.68, 12.2) mm, rotated rx 0 ry 90 rz 0 deg; joints [-11.795, -27.394, 110.238, -15.841, -82.251, 51.177]
  Call Extruder(0.010)
  MoveL 5561 to (509.6, 500.03, 12.2) mm, rotated rx 0 ry 90 rz 0 deg; joints [-11.827, -27.393, 110.229, -15.873, -82.245, 51.183]
  Call Extruder(0.007)
  MoveL 5562 to (509.25, 500.02, 12.2) mm, rotated rx 0 ry 90 rz 0 deg; joints [-11.833, -27.4, 110.272, -15.878, -82.279, 51.174]
  Call Extruder(0.036)
  MoveL 5563 to (508.02, 500.02, 12.2) mm, rotated rx 0 ry 90 rz 0 deg; joints [-11.856, -27.424, 110.42, -15.897, -82.399, 51.142]
  Call Extruder(0.010)
  MoveL 5564 to (507.67, 500.02, 12.2) mm, rotated rx 0 ry 90 rz 0 deg; joints [-11.863, -27.431, 110.462, -15.902, -82.433, 51.133]
  Call Extruder(0.007)
  MoveL 5565 to (507.67, 500.37, 12.2) mm, rotated rx 0 ry 90 rz 0 deg; joints [-11.895, -27.43, 110.453, -15.934, -82.427, 51.139]
  Call Extruder(0.062)
  MoveL 5566 to (507.67, 502.5, 12.2) mm, rotated rx 0 ry 90 rz 0 deg; joints [-12.087, -27.421, 110.399, -16.13, -82.39, 51.175]
  Call Extruder(0.056)
  MoveL 5567 to (509.6, 502.5, 12.2) mm, rotated rx 0 ry 90 rz 0 deg; joints [-12.05, -27.382, 110.166, -16.1, -82.202, 51.225]
  Call Extruder(0.206)
  MoveL 5568 to (509.6, 509.6, 12.2) mm, rotated rx 0 ry 90 rz 0 deg; joints [-12.688, -27.351, 109.979, -16.75, -82.075, 51.347]
  Call Extruder(0.559)
  MoveL 5569 to (490.4, 509.6, 12.2) mm, rotated rx 0 ry 90 rz 0 deg; joints [-13.088, -27.709, 112.266, -17.084, -83.933, 50.825]
  MoveL 5570 to (490.4, 490.4, 12.2) mm, rotated rx 0 ry 90 rz 0 deg; joints [-11.303, -27.779, 112.756, -15.278, -84.292, 50.55]
  Call Extruder(0.182)
  MoveL 5571 to (496.66, 490.4, 12.2) mm, rotated rx 0 ry 90 rz 0 deg; joints [-11.187, -27.672, 112.013, -15.179, -83.675, 50.708]
  Call Extruder(0.010)
  MoveL 5572 to (497.01, 490.4, 12.2) mm, rotated rx 0 ry 90 rz 0 deg; joints [-11.181, -27.666, 111.971, -15.174, -83.64, 50.716]
  Call Extruder(0.007)
  MoveL 5573 to (497.01, 490.75, 12.2) mm, rotated rx 0 ry 90 rz 0 deg; joints [-11.213, -27.665, 111.963, -15.206, -83.634, 50.721]
  Call Extruder(0.045)
  MoveL 5574 to (497.01, 492.3, 12.2) mm, rotated rx 0 ry 90 rz 0 deg; joints [-11.357, -27.66, 111.927, -15.352, -83.608, 50.744]
  Set speed (120.0 mm/s)
  MoveL 5575 to (497.41, 492.3, 12.2) mm, rotated rx 0 ry 90 rz 0 deg; joints [-11.349, -27.652, 111.879, -15.345, -83.569, 50.754]
  Set speed (1000.0 mm/s)
  MoveL 5576 to (497.41, 492.4, 12.2) mm, rotated rx 0 ry 90 rz 0 deg; joints [-11.358, -27.652, 111.877, -15.355, -83.567, 50.755]
  Set speed (1000.0 mm/s)
  MoveL 5577 to (507.28, 499.5, 12.2) mm, rotated rx 0 ry 90 rz 0 deg; joints [-11.822, -27.441, 110.522, -15.86, -82.479, 51.115]
  Set speed (1000.0 mm/s)
  MoveL 5578 to (507.31, 499.46, 12.2) mm, rotated rx 0 ry 90 rz 0 deg; joints [-11.819, -27.44, 110.519, -15.856, -82.477, 51.115]
  Set speed (15.0 mm/s)
  Call Extruder(0.005)
  MoveL 5579 to (507.71, 499.56, 12.2) mm, rotated rx 0 ry 90 rz 0 deg; joints [-11.82, -27.432, 110.469, -15.859, -82.437, 51.127]
  Call Extruder(0.017)
  MoveL 5580 to (509.17, 499.59, 12.2) mm, rotated rx 0 ry 90 rz 0 deg; joints [-11.795, -27.403, 110.293, -15.839, -82.294, 51.164]
  Set speed (120.0 mm/s)
  MoveL 5581 to (508.9, 499.8, 12.2) mm, rotated rx 0 ry 90 rz 0 deg; joints [-11.82, -27.408, 110.319, -15.863, -82.316, 51.161]
  Set speed (1000.0 mm/s)
  MoveL 5582 to (490.68, 490.68, 12.2) mm, rotated rx 0 ry 90 rz 0 deg; joints [-11.324, -27.773, 112.716, -15.3, -84.259, 50.561]
  Set speed (1000.0 mm/s)
  MoveL 5583 to (490.68, 490.68, 12.3) mm, rotated rx 0 ry 90 rz 0 deg; joints [-11.324, -27.784, 112.722, -15.3, -84.254, 50.562]
  Set speed (30.0 mm/s)
  Call Extruder(0.767)
  MoveL 5584 to (509.32, 509.32, 12.3) mm, rotated rx 0 ry 90 rz 0 deg; joints [-12.669, -27.368, 110.025, -16.729, -82.102, 51.337]
  MoveL 5585 to (509.44, 509.44, 12.3) mm, rotated rx 0 ry 90 rz 0 deg; joints [-12.677, -27.365, 110.007, -16.738, -82.088, 51.342]
  Set speed (120.0 mm/s)
  MoveL 5586 to (507.39, 502.51, 12.3) mm, rotated rx 0 ry 90 rz 0 deg; joints [-12.094, -27.437, 110.438, -16.136, -82.412, 51.169]
  Set speed (30.0 mm/s)
  Call Extruder(0.280)
  MoveL 5587 to (500.58, 509.32, 12.3) mm, rotated rx 0 ry 90 rz 0 deg; joints [-12.847, -27.539, 111.072, -16.876, -82.947, 51.102]
  Set speed (120.0 mm/s)
  MoveL 5588 to (499.42, 509.32, 12.3) mm, rotated rx 0 ry 90 rz 0 deg; joints [-12.872, -27.56, 111.21, -16.896, -83.06, 51.07]
  Set speed (30.0 mm/s)
  Call Extruder(0.360)
  MoveL 5589 to (490.68, 500.58, 12.3) mm, rotated rx 0 ry 90 rz 0 deg; joints [-12.247, -27.749, 112.478, -16.233, -84.075, 50.7]
  Set speed (120.0 mm/s)
  MoveL 5590 to (490.68, 499.42, 12.3) mm, rotated rx 0 ry 90 rz 0 deg; joints [-12.139, -27.754, 112.507, -16.124, -84.097, 50.683]
  Set speed (30.0 mm/s)
  Call Extruder(0.282)
  MoveL 5591 to (497.52, 492.58, 12.3) mm, rotated rx 0 ry 90 rz 0 deg; joints [-11.373, -27.66, 111.865, -15.37, -83.548, 50.762]
  MoveL 5592 to (497.64, 492.46, 12.3) mm, rotated rx 0 ry 90 rz 0 deg; joints [-11.359, -27.658, 111.853, -15.356, -83.538, 50.763]
  Set speed (120.0 mm/s)
  MoveL 5593 to (502.41, 492.51, 12.3) mm, rotated rx 0 ry 90 rz 0 deg; joints [-11.277, -27.572, 111.282, -15.288, -83.069, 50.883]
  Set speed (30.0 mm/s)
  Call Extruder(0.205)
  MoveL 5594 to (507.39, 497.49, 12.3) mm, rotated rx 0 ry 90 rz 0 deg; joints [-11.639, -27.457, 110.564, -15.673, -82.498, 51.086]
  MoveL 5595 to (507.51, 497.61, 12.3) mm, rotated rx 0 ry 90 rz 0 deg; joints [-11.647, -27.455, 110.546, -15.683, -82.484, 51.091]
  Set speed (120.0 mm/s)
  MoveL 5596 to (509.32, 490.68, 12.3) mm, rotated rx 0 ry 90 rz 0 deg; joints [-10.985, -27.446, 110.496, -15.017, -82.422, 51.025]
  Set speed (30.0 mm/s)
  Call Extruder(0.767)
  MoveL 5597 to (490.68, 509.32, 12.3) mm, rotated rx 0 ry 90 rz 0 deg; joints [-13.056, -27.716, 112.246, -17.052, -83.907, 50.83]
  MoveL 5598 to (490.56, 509.44, 12.3) mm, rotated rx 0 ry 90 rz 0 deg; joints [-13.07, -27.718, 112.257, -17.066, -83.916, 50.829]
  Set speed (120.0 mm/s)
  MoveL 5599 to (496.89, 492.37, 12.3) mm, rotated rx 0 ry 90 rz 0 deg; joints [-11.365, -27.672, 111.945, -15.36, -83.614, 50.743]
  Set speed (1000.0 mm/s)
  MoveL 5600 to (496.96, 492.3, 12.3) mm, rotated rx 0 ry 90 rz 0 deg; joints [-11.358, -27.671, 111.938, -15.353, -83.608, 50.744]
  Set speed (15.0 mm/s)
  Call Extruder(0.072)
  MoveL 5601 to (499.42, 492.3, 12.3) mm, rotated rx 0 ry 90 rz 0 deg; joints [-11.312, -27.627, 111.645, -15.314, -83.367, 50.805]
  Call Extruder(0.055)
  MoveL 5602 to (499.42, 490.4, 12.3) mm, rotated rx 0 ry 90 rz 0 deg; joints [-11.137, -27.634, 111.69, -15.137, -83.399, 50.778]
  Call Extruder(0.009)
  MoveL 5603 to (499.71, 490.4, 12.3) mm, rotated rx 0 ry 90 rz 0 deg; joints [-11.132, -27.629, 111.655, -15.132, -83.37, 50.785]
  Call Extruder(0.023)
  MoveL 5604 to (499.71, 492.3, 12.3) mm, rotated rx 0 ry 90 rz 0 deg; joints [-11.307, -27.622, 111.61, -15.31, -83.338, 50.813]
  Call Extruder(0.060)
  MoveL 5605 to (501.78, 492.3, 12.3) mm, rotated rx 0 ry 90 rz 0 deg; joints [-11.269, -27.584, 111.363, -15.278, -83.135, 50.865]
  Call Extruder(0.010)
  MoveL 5606 to (502.13, 492.3, 12.3) mm, rotated rx 0 ry 90 rz 0 deg; joints [-11.262, -27.578, 111.321, -15.273, -83.1, 50.873]
  Call Extruder(0.007)
  MoveL 5607 to (502.13, 491.95, 12.3) mm, rotated rx 0 ry 90 rz 0 deg; joints [-11.23, -27.579, 111.329, -15.24, -83.106, 50.868]
  Call Extruder(0.035)
  MoveL 5608 to (502.13, 490.75, 12.3) mm, rotated rx 0 ry 90 rz 0 deg; joints [-11.12, -27.583, 111.358, -15.128, -83.126, 50.85]
  Call Extruder(0.010)
  MoveL 5609 to (502.13, 490.4, 12.3) mm, rotated rx 0 ry 90 rz 0 deg; joints [-11.088, -27.585, 111.366, -15.096, -83.132, 50.845]
  Call Extruder(0.007)
  MoveL 5610 to (502.48, 490.4, 12.3) mm, rotated rx 0 ry 90 rz 0 deg; joints [-11.081, -27.578, 111.324, -15.091, -83.098, 50.853]
  Call Extruder(0.207)
  MoveL 5611 to (509.6, 490.4, 12.3) mm, rotated rx 0 ry 90 rz 0 deg; joints [-10.955, -27.442, 110.468, -14.987, -82.399, 51.027]
  Call Extruder(0.179)
  MoveL 5612 to (509.6, 496.55, 12.3) mm, rotated rx 0 ry 90 rz 0 deg; joints [-11.513, -27.418, 110.321, -15.554, -82.298, 51.127]
  Call Extruder(0.056)
  MoveL 5613 to (507.67, 496.55, 12.3) mm, rotated rx 0 ry 90 rz 0 deg; joints [-11.549, -27.456, 110.554, -15.583, -82.487, 51.078]
  Call Extruder(0.062)
  MoveL 5614 to (507.67, 498.7, 12.3) mm, rotated rx 0 ry 90 rz 0 deg; joints [-11.743, -27.447, 110.5, -15.78, -82.45, 51.113]
  Call Extruder(0.010)
  MoveL 5615 to (507.67, 499.05, 12.3) mm, rotated rx 0 ry 90 rz 0 deg; joints [-11.774, -27.446, 110.492, -15.812, -82.444, 51.119]
  Call Extruder(0.007)
  MoveL 5616 to (508.02, 499.05, 12.3) mm, rotated rx 0 ry 90 rz 0 deg; joints [-11.768, -27.439, 110.449, -15.807, -82.41, 51.128]
  Call Extruder(0.036)
  MoveL 5617 to (509.25, 499.05, 12.3) mm, rotated rx 0 ry 90 rz 0 deg; joints [-11.745, -27.414, 110.301, -15.788, -82.29, 51.159]
  Call Extruder(0.010)
  MoveL 5618 to (509.6, 499.05, 12.3) mm, rotated rx 0 ry 90 rz 0 deg; joints [-11.738, -27.407, 110.259, -15.783, -82.256, 51.168]
  Call Extruder(0.007)
  MoveL 5619 to (509.6, 499.39, 12.3) mm, rotated rx 0 ry 90 rz 0 deg; joints [-11.77, -27.406, 110.25, -15.815, -82.25, 51.174]
  Call Extruder(0.010)
  MoveL 5620 to (509.6, 499.73, 12.3) mm, rotated rx 0 ry 90 rz 0 deg; joints [-11.8, -27.404, 110.242, -15.846, -82.244, 51.179]
  Call Extruder(0.010)
  MoveL 5621 to (509.6, 500.08, 12.3) mm, rotated rx 0 ry 90 rz 0 deg; joints [-11.832, -27.403, 110.233, -15.878, -82.238, 51.185]
  Call Extruder(0.007)
  MoveL 5622 to (509.25, 500.08, 12.3) mm, rotated rx 0 ry 90 rz 0 deg; joints [-11.838, -27.41, 110.275, -15.883, -82.273, 51.176]
  Call Extruder(0.036)
  MoveL 5623 to (508.02, 500.08, 12.3) mm, rotated rx 0 ry 90 rz 0 deg; joints [-11.861, -27.434, 110.424, -15.902, -82.393, 51.145]
  Call Extruder(0.010)
  MoveL 5624 to (507.67, 500.08, 12.3) mm, rotated rx 0 ry 90 rz 0 deg; joints [-11.868, -27.441, 110.466, -15.908, -82.427, 51.136]
  Call Extruder(0.007)
  MoveL 5625 to (507.67, 500.43, 12.3) mm, rotated rx 0 ry 90 rz 0 deg; joints [-11.9, -27.44, 110.457, -15.94, -82.421, 51.142]
  Call Extruder(0.062)
  MoveL 5626 to (507.67, 502.56, 12.3) mm, rotated rx 0 ry 90 rz 0 deg; joints [-12.092, -27.431, 110.403, -16.136, -82.383, 51.177]
  Call Extruder(0.056)
  MoveL 5627 to (509.6, 502.56, 12.3) mm, rotated rx 0 ry 90 rz 0 deg; joints [-12.055, -27.392, 110.17, -16.106, -82.195, 51.227]
  Call Extruder(0.205)
  MoveL 5628 to (509.6, 509.6, 12.3) mm, rotated rx 0 ry 90 rz 0 deg; joints [-12.688, -27.361, 109.984, -16.75, -82.07, 51.349]
  Call Extruder(0.559)
  MoveL 5629 to (490.4, 509.6, 12.3) mm, rotated rx 0 ry 90 rz 0 deg; joints [-13.088, -27.72, 112.271, -17.084, -83.928, 50.827]
  MoveL 5630 to (490.4, 490.4, 12.3) mm, rotated rx 0 ry 90 rz 0 deg; joints [-11.303, -27.789, 112.761, -15.278, -84.286, 50.551]
  Call Extruder(0.181)
  MoveL 5631 to (496.61, 490.4, 12.3) mm, rotated rx 0 ry 90 rz 0 deg; joints [-11.188, -27.684, 112.025, -15.18, -83.675, 50.708]
  Call Extruder(0.010)
  MoveL 5632 to (496.96, 490.4, 12.3) mm, rotated rx 0 ry 90 rz 0 deg; joints [-11.182, -27.678, 111.983, -15.175, -83.641, 50.716]
  Call Extruder(0.007)
  MoveL 5633 to (496.96, 490.75, 12.3) mm, rotated rx 0 ry 90 rz 0 deg; joints [-11.214, -27.677, 111.975, -15.207, -83.635, 50.721]
  Call Extruder(0.045)
  MoveL 5634 to (496.96, 492.3, 12.3) mm, rotated rx 0 ry 90 rz 0 deg; joints [-11.358, -27.671, 111.938, -15.353, -83.608, 50.744]
  Set speed (120.0 mm/s)
  MoveL 5635 to (497.36, 492.3, 12.3) mm, rotated rx 0 ry 90 rz 0 deg; joints [-11.35, -27.664, 111.891, -15.346, -83.569, 50.754]
  Set speed (1000.0 mm/s)
  MoveL 5636 to (497.36, 492.4, 12.3) mm, rotated rx 0 ry 90 rz 0 deg; joints [-11.359, -27.664, 111.888, -15.356, -83.567, 50.755]
  Set speed (1000.0 mm/s)
  MoveL 5637 to (507.3, 499.38, 12.3) mm, rotated rx 0 ry 90 rz 0 deg; joints [-11.811, -27.452, 110.528, -15.849, -82.475, 51.115]
  Set speed (1000.0 mm/s)
  MoveL 5638 to (507.48, 499.56, 12.3) mm, rotated rx 0 ry 90 rz 0 deg; joints [-11.825, -27.447, 110.501, -15.863, -82.454, 51.122]
  Set speed (15.0 mm/s)
  Call Extruder(0.011)
  MoveL 5639 to (507.98, 499.56, 12.3) mm, rotated rx 0 ry 90 rz 0 deg; joints [-11.815, -27.437, 110.442, -15.855, -82.406, 51.135]
  Call Extruder(0.022)
  MoveL 5640 to (508.97, 499.56, 12.3) mm, rotated rx 0 ry 90 rz 0 deg; joints [-11.797, -27.418, 110.323, -15.84, -82.309, 51.16]
  Set speed (120.0 mm/s)
  MoveL 5641 to (509.15, 499.75, 12.3) mm, rotated rx 0 ry 90 rz 0 deg; joints [-11.81, -27.413, 110.295, -15.854, -82.288, 51.168]
  Set speed (1000.0 mm/s)
  MoveL 5642 to (490.68, 490.68, 12.3) mm, rotated rx 0 ry 90 rz 0 deg; joints [-11.324, -27.784, 112.722, -15.3, -84.254, 50.562]
  Set speed (1000.0 mm/s)
  MoveL 5643 to (490.68, 490.68, 12.4) mm, rotated rx 0 ry 90 rz 0 deg; joints [-11.324, -27.794, 112.727, -15.3, -84.249, 50.564]
  Set speed (30.0 mm/s)
  Call Extruder(0.767)
  MoveL 5644 to (509.32, 509.32, 12.4) mm, rotated rx 0 ry 90 rz 0 deg; joints [-12.669, -27.379, 110.03, -16.729, -82.097, 51.338]
  MoveL 5645 to (509.44, 509.44, 12.4) mm, rotated rx 0 ry 90 rz 0 deg; joints [-12.677, -27.376, 110.012, -16.738, -82.083, 51.344]
  Set speed (120.0 mm/s)
  MoveL 5646 to (507.39, 502.51, 12.4) mm, rotated rx 0 ry 90 rz 0 deg; joints [-12.094, -27.447, 110.443, -16.136, -82.406, 51.17]
  Set speed (30.0 mm/s)
  Call Extruder(0.280)
  MoveL 5647 to (500.58, 509.32, 12.4) mm, rotated rx 0 ry 90 rz 0 deg; joints [-12.847, -27.549, 111.077, -16.876, -82.942, 51.103]
  Set speed (120.0 mm/s)
  MoveL 5648 to (499.42, 509.32, 12.4) mm, rotated rx 0 ry 90 rz 0 deg; joints [-12.872, -27.571, 111.216, -16.896, -83.054, 51.072]
  Set speed (30.0 mm/s)
  Call Extruder(0.360)
  MoveL 5649 to (490.68, 500.58, 12.4) mm, rotated rx 0 ry 90 rz 0 deg; joints [-12.247, -27.76, 112.483, -16.233, -84.07, 50.701]
  Set speed (120.0 mm/s)
  MoveL 5650 to (490.68, 499.42, 12.4) mm, rotated rx 0 ry 90 rz 0 deg; joints [-12.139, -27.764, 112.512, -16.124, -84.091, 50.685]
  Set speed (30.0 mm/s)
  Call Extruder(0.282)
  MoveL 5651 to (497.52, 492.58, 12.4) mm, rotated rx 0 ry 90 rz 0 deg; joints [-11.373, -27.671, 111.87, -15.37, -83.543, 50.763]
  MoveL 5652 to (497.64, 492.46, 12.4) mm, rotated rx 0 ry 90 rz 0 deg; joints [-11.359, -27.669, 111.858, -15.357, -83.533, 50.765]
  Set speed (120.0 mm/s)
  MoveL 5653 to (502.47, 492.58, 12.4) mm, rotated rx 0 ry 90 rz 0 deg; joints [-11.281, -27.581, 111.278, -15.293, -83.057, 50.887]
  Set speed (30.0 mm/s)
  Call Extruder(0.202)
  MoveL 5654 to (507.39, 497.49, 12.4) mm, rotated rx 0 ry 90 rz 0 deg; joints [-11.639, -27.468, 110.569, -15.674, -82.493, 51.088]
  MoveL 5655 to (507.51, 497.61, 12.4) mm, rotated rx 0 ry 90 rz 0 deg; joints [-11.647, -27.465, 110.552, -15.683, -82.479, 51.093]
  Set speed (120.0 mm/s)
  MoveL 5656 to (509.32, 490.68, 12.4) mm, rotated rx 0 ry 90 rz 0 deg; joints [-10.985, -27.457, 110.501, -15.017, -82.417, 51.026]
  Set speed (30.0 mm/s)
  Call Extruder(0.767)
  MoveL 5657 to (490.68, 509.32, 12.4) mm, rotated rx 0 ry 90 rz 0 deg; joints [-13.056, -27.727, 112.251, -17.052, -83.901, 50.832]
  MoveL 5658 to (490.56, 509.44, 12.4) mm, rotated rx 0 ry 90 rz 0 deg; joints [-13.07, -27.728, 112.262, -17.066, -83.911, 50.83]
  Set speed (120.0 mm/s)
  MoveL 5659 to (502.27, 492.37, 12.4) mm, rotated rx 0 ry 90 rz 0 deg; joints [-11.266, -27.585, 111.308, -15.277, -83.081, 50.879]
  Set speed (1000.0 mm/s)
  MoveL 5660 to (502.2, 492.3, 12.4) mm, rotated rx 0 ry 90 rz 0 deg; joints [-11.261, -27.587, 111.318, -15.272, -83.089, 50.876]
  Set speed (15.0 mm/s)
  Call Extruder(0.010)
  MoveL 5661 to (502.2, 491.95, 12.4) mm, rotated rx 0 ry 90 rz 0 deg; joints [-11.229, -27.588, 111.327, -15.239, -83.095, 50.871]
  Call Extruder(0.035)
  MoveL 5662 to (502.19, 490.75, 12.4) mm, rotated rx 0 ry 90 rz 0 deg; joints [-11.119, -27.593, 111.355, -15.128, -83.115, 50.853]
  Call Extruder(0.010)
  MoveL 5663 to (502.2, 490.4, 12.4) mm, rotated rx 0 ry 90 rz 0 deg; joints [-11.087, -27.594, 111.363, -15.095, -83.121, 50.848]
  Call Extruder(0.007)
  MoveL 5664 to (502.55, 490.4, 12.4) mm, rotated rx 0 ry 90 rz 0 deg; joints [-11.08, -27.587, 111.322, -15.09, -83.086, 50.856]
  Call Extruder(0.205)
  MoveL 5665 to (509.6, 490.4, 12.4) mm, rotated rx 0 ry 90 rz 0 deg; joints [-10.955, -27.452, 110.473, -14.987, -82.394, 51.029]
  Call Extruder(0.177)
  MoveL 5666 to (509.6, 496.49, 12.4) mm, rotated rx 0 ry 90 rz 0 deg; joints [-11.507, -27.428, 110.328, -15.548, -82.294, 51.127]
  Call Extruder(0.056)
  MoveL 5667 to (507.67, 496.49, 12.4) mm, rotated rx 0 ry 90 rz 0 deg; joints [-11.543, -27.466, 110.56, -15.578, -82.483, 51.079]
  Call Extruder(0.073)
  MoveL 5668 to (507.67, 498.99, 12.4) mm, rotated rx 0 ry 90 rz 0 deg; joints [-11.769, -27.456, 110.498, -15.807, -82.44, 51.119]
  Call Extruder(0.056)
  MoveL 5669 to (509.6, 498.99, 12.4) mm, rotated rx 0 ry 90 rz 0 deg; joints [-11.733, -27.418, 110.266, -15.778, -82.252, 51.168]
  Call Extruder(0.023)
  MoveL 5670 to (509.6, 499.79, 12.4) mm, rotated rx 0 ry 90 rz 0 deg; joints [-11.805, -27.415, 110.246, -15.851, -82.238, 51.182]
  Call Extruder(0.010)
  MoveL 5671 to (509.6, 500.14, 12.4) mm, rotated rx 0 ry 90 rz 0 deg; joints [-11.837, -27.413, 110.237, -15.883, -82.232, 51.188]
  Call Extruder(0.007)
  MoveL 5672 to (509.25, 500.14, 12.4) mm, rotated rx 0 ry 90 rz 0 deg; joints [-11.843, -27.42, 110.279, -15.889, -82.266, 51.179]
  Call Extruder(0.036)
  MoveL 5673 to (508.02, 500.14, 12.4) mm, rotated rx 0 ry 90 rz 0 deg; joints [-11.867, -27.445, 110.427, -15.908, -82.386, 51.147]
  Call Extruder(0.010)
  MoveL 5674 to (507.67, 500.13, 12.4) mm, rotated rx 0 ry 90 rz 0 deg; joints [-11.873, -27.452, 110.47, -15.913, -82.421, 51.138]
  Call Extruder(0.007)
  MoveL 5675 to (507.67, 500.49, 12.4) mm, rotated rx 0 ry 90 rz 0 deg; joints [-11.905, -27.45, 110.461, -15.945, -82.414, 51.144]
  Call Extruder(0.062)
  MoveL 5676 to (507.67, 502.62, 12.4) mm, rotated rx 0 ry 90 rz 0 deg; joints [-12.098, -27.441, 110.406, -16.141, -82.377, 51.179]
  Call Extruder(0.056)
  MoveL 5677 to (509.6, 502.62, 12.4) mm, rotated rx 0 ry 90 rz 0 deg; joints [-12.061, -27.403, 110.173, -16.111, -82.189, 51.229]
  Call Extruder(0.203)
  MoveL 5678 to (509.6, 509.6, 12.4) mm, rotated rx 0 ry 90 rz 0 deg; joints [-12.688, -27.372, 109.989, -16.75, -82.065, 51.351]
  Call Extruder(0.559)
  MoveL 5679 to (490.4, 509.6, 12.4) mm, rotated rx 0 ry 90 rz 0 deg; joints [-13.088, -27.73, 112.276, -17.084, -83.923, 50.828]
  MoveL 5680 to (490.4, 490.4, 12.4) mm, rotated rx 0 ry 90 rz 0 deg; joints [-11.303, -27.8, 112.766, -15.278, -84.281, 50.553]
  Call Extruder(0.189)
  MoveL 5681 to (496.9, 490.4, 12.4) mm, rotated rx 0 ry 90 rz 0 deg; joints [-11.183, -27.689, 111.995, -15.176, -83.641, 50.716]
  Call Extruder(0.055)
  MoveL 5682 to (496.9, 492.3, 12.4) mm, rotated rx 0 ry 90 rz 0 deg; joints [-11.359, -27.683, 111.95, -15.354, -83.609, 50.744]
  Call Extruder(0.072)
  MoveL 5683 to (499.36, 492.3, 12.4) mm, rotated rx 0 ry 90 rz 0 deg; joints [-11.313, -27.639, 111.657, -15.315, -83.367, 50.805]
  Call Extruder(0.055)
  MoveL 5684 to (499.36, 490.4, 12.4) mm, rotated rx 0 ry 90 rz 0 deg; joints [-11.138, -27.646, 111.702, -15.138, -83.399, 50.778]
  Call Extruder(0.012)
  MoveL 5685 to (499.78, 490.4, 12.4) mm, rotated rx 0 ry 90 rz 0 deg; joints [-11.13, -27.638, 111.653, -15.132, -83.358, 50.788]
  Call Extruder(0.033)
  MoveL 5686 to (499.78, 492.3, 12.4) mm, rotated rx 0 ry 90 rz 0 deg; joints [-11.305, -27.631, 111.607, -15.309, -83.326, 50.816]
  Call Extruder(0.060)
  MoveL 5687 to (501.85, 492.3, 12.4) mm, rotated rx 0 ry 90 rz 0 deg; joints [-11.267, -27.593, 111.36, -15.277, -83.123, 50.868]
  Call Extruder(0.007)
  MoveL 5688 to (502.2, 492.3, 12.4) mm, rotated rx 0 ry 90 rz 0 deg; joints [-11.261, -27.587, 111.318, -15.272, -83.089, 50.876]
  Set speed (120.0 mm/s)
  MoveL 5689 to (502.2, 491.95, 12.4) mm, rotated rx 0 ry 90 rz 0 deg; joints [-11.229, -27.588, 111.327, -15.239, -83.095, 50.871]
  Set speed (1000.0 mm/s)
  MoveL 5690 to (502.2, 491.9, 12.4) mm, rotated rx 0 ry 90 rz 0 deg; joints [-11.224, -27.588, 111.328, -15.235, -83.096, 50.87]
  Set speed (1000.0 mm/s)
  MoveL 5691 to (502.3, 491.9, 12.4) mm, rotated rx 0 ry 90 rz 0 deg; joints [-11.222, -27.587, 111.316, -15.233, -83.086, 50.873]
  Set speed (1000.0 mm/s)
  MoveL 5692 to (507.46, 499.32, 12.4) mm, rotated rx 0 ry 90 rz 0 deg; joints [-11.803, -27.459, 110.515, -15.841, -82.455, 51.119]
  Set speed (1000.0 mm/s)
  MoveL 5693 to (507.37, 499.41, 12.4) mm, rotated rx 0 ry 90 rz 0 deg; joints [-11.813, -27.46, 110.523, -15.85, -82.462, 51.119]
  Set speed (15.0 mm/s)
  Call Extruder(0.008)
  MoveL 5694 to (507.71, 499.56, 12.4) mm, rotated rx 0 ry 90 rz 0 deg; joints [-11.82, -27.453, 110.479, -15.859, -82.426, 51.13]
  Call Extruder(0.032)
  MoveL 5695 to (509.11, 499.65, 12.4) mm, rotated rx 0 ry 90 rz 0 deg; joints [-11.802, -27.425, 110.308, -15.846, -82.289, 51.167]
  Set speed (120.0 mm/s)
  MoveL 5696 to (508.95, 499.69, 12.4) mm, rotated rx 0 ry 90 rz 0 deg; joints [-11.808, -27.428, 110.326, -15.852, -82.303, 51.163]
  Set speed (1000.0 mm/s)
  MoveL 5697 to (490.68, 490.68, 12.4) mm, rotated rx 0 ry 90 rz 0 deg; joints [-11.324, -27.794, 112.727, -15.3, -84.249, 50.564]
  Set speed (1000.0 mm/s)
  MoveL 5698 to (490.68, 490.68, 12.5) mm, rotated rx 0 ry 90 rz 0 deg; joints [-11.324, -27.805, 112.732, -15.3, -84.244, 50.565]
  Set speed (30.0 mm/s)
  Call Extruder(0.767)
  MoveL 5699 to (509.32, 509.32, 12.5) mm, rotated rx 0 ry 90 rz 0 deg; joints [-12.669, -27.389, 110.036, -16.729, -82.092, 51.34]
  MoveL 5700 to (509.44, 509.44, 12.5) mm, rotated rx 0 ry 90 rz 0 deg; joints [-12.677, -27.386, 110.017, -16.739, -82.078, 51.345]
  Set speed (120.0 mm/s)
  MoveL 5701 to (507.38, 502.51, 12.5) mm, rotated rx 0 ry 90 rz 0 deg; joints [-12.094, -27.458, 110.448, -16.136, -82.401, 51.172]
  Set speed (30.0 mm/s)
  Call Extruder(0.280)
  MoveL 5702 to (500.58, 509.32, 12.5) mm, rotated rx 0 ry 90 rz 0 deg; joints [-12.847, -27.56, 111.083, -16.876, -82.937, 51.105]
  Set speed (120.0 mm/s)
  MoveL 5703 to (499.42, 509.32, 12.5) mm, rotated rx 0 ry 90 rz 0 deg; joints [-12.872, -27.581, 111.221, -16.896, -83.049, 51.073]
  Set speed (30.0 mm/s)
  Call Extruder(0.360)
  MoveL 5704 to (490.68, 500.58, 12.5) mm, rotated rx 0 ry 90 rz 0 deg; joints [-12.247, -27.771, 112.488, -16.233, -84.064, 50.703]
  Set speed (120.0 mm/s)
  MoveL 5705 to (490.68, 499.42, 12.5) mm, rotated rx 0 ry 90 rz 0 deg; joints [-12.139, -27.775, 112.518, -16.124, -84.086, 50.686]
  Set speed (30.0 mm/s)
  Call Extruder(0.282)
  MoveL 5706 to (497.52, 492.58, 12.5) mm, rotated rx 0 ry 90 rz 0 deg; joints [-11.373, -27.681, 111.875, -15.37, -83.538, 50.765]
  MoveL 5707 to (497.64, 492.46, 12.5) mm, rotated rx 0 ry 90 rz 0 deg; joints [-11.359, -27.68, 111.863, -15.357, -83.528, 50.766]
  Set speed (120.0 mm/s)
  MoveL 5708 to (502.48, 492.58, 12.5) mm, rotated rx 0 ry 90 rz 0 deg; joints [-11.281, -27.591, 111.283, -15.294, -83.051, 50.889]
  Set speed (30.0 mm/s)
  Call Extruder(0.202)
  MoveL 5709 to (507.39, 497.49, 12.5) mm, rotated rx 0 ry 90 rz 0 deg; joints [-11.639, -27.478, 110.575, -15.674, -82.488, 51.089]
  MoveL 5710 to (507.51, 497.61, 12.5) mm, rotated rx 0 ry 90 rz 0 deg; joints [-11.647, -27.476, 110.557, -15.683, -82.474, 51.094]
  Set speed (120.0 mm/s)
  MoveL 5711 to (509.32, 490.68, 12.5) mm, rotated rx 0 ry 90 rz 0 deg; joints [-10.985, -27.467, 110.506, -15.017, -82.412, 51.028]
  Set speed (30.0 mm/s)
  Call Extruder(0.767)
  MoveL 5712 to (490.68, 509.32, 12.5) mm, rotated rx 0 ry 90 rz 0 deg; joints [-13.056, -27.737, 112.256, -17.053, -83.896, 50.833]
  MoveL 5713 to (490.56, 509.44, 12.5) mm, rotated rx 0 ry 90 rz 0 deg; joints [-13.07, -27.739, 112.268, -17.066, -83.906, 50.832]
  Set speed (120.0 mm/s)
  MoveL 5714 to (502.33, 492.37, 12.5) mm, rotated rx 0 ry 90 rz 0 deg; joints [-11.265, -27.595, 111.306, -15.276, -83.069, 50.882]
  Set speed (1000.0 mm/s)
  MoveL 5715 to (502.26, 492.3, 12.5) mm, rotated rx 0 ry 90 rz 0 deg; joints [-11.26, -27.596, 111.316, -15.271, -83.077, 50.879]
  Set speed (15.0 mm/s)
  Call Extruder(0.010)
  MoveL 5716 to (502.26, 491.95, 12.5) mm, rotated rx 0 ry 90 rz 0 deg; joints [-11.228, -27.598, 111.324, -15.238, -83.083, 50.874]
  Call Extruder(0.035)
  MoveL 5717 to (502.26, 490.75, 12.5) mm, rotated rx 0 ry 90 rz 0 deg; joints [-11.118, -27.602, 111.353, -15.127, -83.103, 50.856]
  Call Extruder(0.010)
  MoveL 5718 to (502.26, 490.4, 12.5) mm, rotated rx 0 ry 90 rz 0 deg; joints [-11.085, -27.603, 111.361, -15.094, -83.109, 50.851]
  Call Extruder(0.007)
